Fanuc TP program (LS listing): 190220_hosenrohr_oV3.ls

/PROG  190220_hosenrohr_oV3
/ATTR
COMMENT	= "19-02-22 10:03:29";
PROG_SIZE	= 0;
DEFAULT_GROUP	= 1, 1, *, *, *;
/APPL
    ARC Welding Equipment: 1, *, *, *, *;
/MN
   1:  CALL HOME_ALL;
   1:  UFRAME_NUM = 1;
   1:  UTOOL_NUM = 3;
   1:  COL GUARD ADJUST 150;
   1:  ! -- Layer/Ebene 97 -- !;
   1:  PR[91] = PR[90];
   1:  PR[GP1:91,1] = PR[GP1:90,1] + 0.151;
   1:  PR[GP1:91,2] = PR[GP1:90,2] + 28.908;
   1:  PR[GP1:91,3] = PR[GP1:90,3] + 59.475;
   1:  !Sicherheitspunkt!;
   1:  PR[92] = PR[91];
   1:  PR[92] = PR[GP1:92,3] + 50;
   1:J PR[92];
   1:  !Schweissanfang anfahren!;
   1:L PR[91] R[100]mm/sec CNT100;
   1:  CALL LASER_DRAHT_START;
   1:  PR[GP1:91,1] = PR[GP1:90,1] + -2.869;
   1:  PR[GP1:91,2] = PR[GP1:90,2] + 29.610;
   1:L PR[91] R[100]mm/sec CNT100;
   1:  PR[GP1:91,1] = PR[GP1:90,1] + -5.863;
   1:  PR[GP1:91,2] = PR[GP1:90,2] + 31.726;
   1:L PR[91] R[100]mm/sec CNT100;
   1:  PR[GP1:91,1] = PR[GP1:90,1] + -7.882;
   1:  PR[GP1:91,2] = PR[GP1:90,2] + 32.782;
   1:L PR[91] R[100]mm/sec CNT100;
   1:  PR[GP1:91,1] = PR[GP1:90,1] + -10.388;
   1:  PR[GP1:91,2] = PR[GP1:90,2] + 33.587;
   1:L PR[91] R[100]mm/sec CNT100;
   1:  PR[GP1:91,1] = PR[GP1:90,1] + -18.640;
   1:  PR[GP1:91,2] = PR[GP1:90,2] + 36.440;
   1:L PR[91] R[100]mm/sec CNT100;
   1:  PR[GP1:91,1] = PR[GP1:90,1] + -21.584;
   1:  PR[GP1:91,2] = PR[GP1:90,2] + 36.825;
   1:L PR[91] R[100]mm/sec CNT100;
   1:  PR[GP1:91,1] = PR[GP1:90,1] + -25.063;
   1:  PR[GP1:91,2] = PR[GP1:90,2] + 36.705;
   1:L PR[91] R[100]mm/sec CNT100;
   1:  PR[GP1:91,1] = PR[GP1:90,1] + -32.430;
   1:  PR[GP1:91,2] = PR[GP1:90,2] + 36.668;
   1:L PR[91] R[100]mm/sec CNT100;
   1:  PR[GP1:91,1] = PR[GP1:90,1] + -36.082;
   1:  PR[GP1:91,2] = PR[GP1:90,2] + 35.880;
   1:L PR[91] R[100]mm/sec CNT100;
   1:  PR[GP1:91,1] = PR[GP1:90,1] + -40.103;
   1:  PR[GP1:91,2] = PR[GP1:90,2] + 34.289;
   1:L PR[91] R[100]mm/sec CNT100;
   1:  PR[GP1:91,1] = PR[GP1:90,1] + -45.491;
   1:  PR[GP1:91,2] = PR[GP1:90,2] + 32.375;
   1:L PR[91] R[100]mm/sec CNT100;
   1:  PR[GP1:91,1] = PR[GP1:90,1] + -49.284;
   1:  PR[GP1:91,2] = PR[GP1:90,2] + 30.013;
   1:L PR[91] R[100]mm/sec CNT100;
   1:  PR[GP1:91,1] = PR[GP1:90,1] + -52.981;
   1:  PR[GP1:91,2] = PR[GP1:90,2] + 26.730;
   1:L PR[91] R[100]mm/sec CNT100;
   1:  PR[GP1:91,1] = PR[GP1:90,1] + -56.222;
   1:  PR[GP1:91,2] = PR[GP1:90,2] + 24.107;
   1:L PR[91] R[100]mm/sec CNT100;
   1:  PR[GP1:91,1] = PR[GP1:90,1] + -59.230;
   1:  PR[GP1:91,2] = PR[GP1:90,2] + 20.191;
   1:L PR[91] R[100]mm/sec CNT100;
   1:  PR[GP1:91,1] = PR[GP1:90,1] + -61.763;
   1:  PR[GP1:91,2] = PR[GP1:90,2] + 15.278;
   1:L PR[91] R[100]mm/sec CNT100;
   1:  PR[GP1:91,1] = PR[GP1:90,1] + -63.337;
   1:  PR[GP1:91,2] = PR[GP1:90,2] + 12.647;
   1:L PR[91] R[100]mm/sec CNT100;
   1:  PR[GP1:91,1] = PR[GP1:90,1] + -64.791;
   1:  PR[GP1:91,2] = PR[GP1:90,2] + 7.718;
   1:L PR[91] R[100]mm/sec CNT100;
   1:  PR[GP1:91,1] = PR[GP1:90,1] + -65.271;
   1:  PR[GP1:91,2] = PR[GP1:90,2] + 2.470;
   1:L PR[91] R[100]mm/sec CNT100;
   1:  PR[GP1:91,1] = PR[GP1:90,1] + -65.744;
   1:  PR[GP1:91,2] = PR[GP1:90,2] + -0.100;
   1:L PR[91] R[100]mm/sec CNT100;
   1:  PR[GP1:91,1] = PR[GP1:90,1] + -65.280;
   1:  PR[GP1:91,2] = PR[GP1:90,2] + -5.239;
   1:L PR[91] R[100]mm/sec CNT100;
   1:  PR[GP1:91,1] = PR[GP1:90,1] + -64.798;
   1:  PR[GP1:91,2] = PR[GP1:90,2] + -7.836;
   1:L PR[91] R[100]mm/sec CNT100;
   1:  PR[GP1:91,1] = PR[GP1:90,1] + -63.331;
   1:  PR[GP1:91,2] = PR[GP1:90,2] + -12.812;
   1:L PR[91] R[100]mm/sec CNT100;
   1:  PR[GP1:91,1] = PR[GP1:90,1] + -60.959;
   1:  PR[GP1:91,2] = PR[GP1:90,2] + -17.463;
   1:L PR[91] R[100]mm/sec CNT100;
   1:  PR[GP1:91,1] = PR[GP1:90,1] + -59.241;
   1:  PR[GP1:91,2] = PR[GP1:90,2] + -20.321;
   1:L PR[91] R[100]mm/sec CNT100;
   1:  PR[GP1:91,1] = PR[GP1:90,1] + -56.211;
   1:  PR[GP1:91,2] = PR[GP1:90,2] + -24.265;
   1:L PR[91] R[100]mm/sec CNT100;
   1:  PR[GP1:91,1] = PR[GP1:90,1] + -52.808;
   1:  PR[GP1:91,2] = PR[GP1:90,2] + -27.318;
   1:L PR[91] R[100]mm/sec CNT100;
   1:  PR[GP1:91,1] = PR[GP1:90,1] + -49.292;
   1:  PR[GP1:91,2] = PR[GP1:90,2] + -30.151;
   1:L PR[91] R[100]mm/sec CNT100;
   1:  PR[GP1:91,1] = PR[GP1:90,1] + -45.477;
   1:  PR[GP1:91,2] = PR[GP1:90,2] + -32.528;
   1:L PR[91] R[100]mm/sec CNT100;
   1:  PR[GP1:91,1] = PR[GP1:90,1] + -41.746;
   1:  PR[GP1:91,2] = PR[GP1:90,2] + -34.026;
   1:L PR[91] R[100]mm/sec CNT100;
   1:  PR[GP1:91,1] = PR[GP1:90,1] + -36.085;
   1:  PR[GP1:91,2] = PR[GP1:90,2] + -36.024;
   1:L PR[91] R[100]mm/sec CNT100;
   1:  PR[GP1:91,1] = PR[GP1:90,1] + -32.412;
   1:  PR[GP1:91,2] = PR[GP1:90,2] + -36.816;
   1:L PR[91] R[100]mm/sec CNT100;
   1:  PR[GP1:91,1] = PR[GP1:90,1] + -29.081;
   1:  PR[GP1:91,2] = PR[GP1:90,2] + -36.944;
   1:L PR[91] R[100]mm/sec CNT100;
   1:  PR[GP1:91,1] = PR[GP1:90,1] + -21.580;
   1:  PR[GP1:91,2] = PR[GP1:90,2] + -36.968;
   1:L PR[91] R[100]mm/sec CNT100;
   1:  PR[GP1:91,1] = PR[GP1:90,1] + -18.619;
   1:  PR[GP1:91,2] = PR[GP1:90,2] + -36.581;
   1:L PR[91] R[100]mm/sec CNT100;
   1:  PR[GP1:91,1] = PR[GP1:90,1] + -16.078;
   1:  PR[GP1:91,2] = PR[GP1:90,2] + -35.772;
   1:L PR[91] R[100]mm/sec CNT100;
   1:  PR[GP1:91,1] = PR[GP1:90,1] + -7.875;
   1:  PR[GP1:91,2] = PR[GP1:90,2] + -32.922;
   1:L PR[91] R[100]mm/sec CNT100;
   1:  PR[GP1:91,1] = PR[GP1:90,1] + -5.858;
   1:  PR[GP1:91,2] = PR[GP1:90,2] + -31.867;
   1:L PR[91] R[100]mm/sec CNT100;
   1:  PR[GP1:91,1] = PR[GP1:90,1] + -2.826;
   1:  PR[GP1:91,2] = PR[GP1:90,2] + -29.664;
   1:L PR[91] R[100]mm/sec CNT100;
   1:  PR[GP1:91,1] = PR[GP1:90,1] + -1.739;
   1:  PR[GP1:91,2] = PR[GP1:90,2] + -29.620;
   1:L PR[91] R[100]mm/sec CNT100;
   1:  PR[GP1:91,1] = PR[GP1:90,1] + 1.633;
   1:  PR[GP1:91,2] = PR[GP1:90,2] + -28.901;
   1:L PR[91] R[100]mm/sec CNT100;
   1:  PR[GP1:91,1] = PR[GP1:90,1] + 1.930;
   1:  PR[GP1:91,2] = PR[GP1:90,2] + -29.139;
   1:L PR[91] R[100]mm/sec CNT100;
   1:  PR[GP1:91,1] = PR[GP1:90,1] + 3.140;
   1:  PR[GP1:91,2] = PR[GP1:90,2] + -29.742;
   1:L PR[91] R[100]mm/sec CNT100;
   1:  PR[GP1:91,1] = PR[GP1:90,1] + 6.073;
   1:  PR[GP1:91,2] = PR[GP1:90,2] + -31.873;
   1:L PR[91] R[100]mm/sec CNT100;
   1:  PR[GP1:91,1] = PR[GP1:90,1] + 8.070;
   1:  PR[GP1:91,2] = PR[GP1:90,2] + -32.915;
   1:L PR[91] R[100]mm/sec CNT100;
   1:  PR[GP1:91,1] = PR[GP1:90,1] + 10.573;
   1:  PR[GP1:91,2] = PR[GP1:90,2] + -33.719;
   1:L PR[91] R[100]mm/sec CNT100;
   1:  PR[GP1:91,1] = PR[GP1:90,1] + 18.836;
   1:  PR[GP1:91,2] = PR[GP1:90,2] + -36.580;
   1:L PR[91] R[100]mm/sec CNT100;
   1:  PR[GP1:91,1] = PR[GP1:90,1] + 21.776;
   1:  PR[GP1:91,2] = PR[GP1:90,2] + -36.966;
   1:L PR[91] R[100]mm/sec CNT100;
   1:  PR[GP1:91,1] = PR[GP1:90,1] + 25.238;
   1:  PR[GP1:91,2] = PR[GP1:90,2] + -36.850;
   1:L PR[91] R[100]mm/sec CNT100;
   1:  PR[GP1:91,1] = PR[GP1:90,1] + 32.611;
   1:  PR[GP1:91,2] = PR[GP1:90,2] + -36.818;
   1:L PR[91] R[100]mm/sec CNT100;
   1:  PR[GP1:91,1] = PR[GP1:90,1] + 36.258;
   1:  PR[GP1:91,2] = PR[GP1:90,2] + -36.033;
   1:L PR[91] R[100]mm/sec CNT100;
   1:  PR[GP1:91,1] = PR[GP1:90,1] + 40.284;
   1:  PR[GP1:91,2] = PR[GP1:90,2] + -34.446;
   1:L PR[91] R[100]mm/sec CNT100;
   1:  PR[GP1:91,1] = PR[GP1:90,1] + 45.678;
   1:  PR[GP1:91,2] = PR[GP1:90,2] + -32.535;
   1:L PR[91] R[100]mm/sec CNT100;
   1:  PR[GP1:91,1] = PR[GP1:90,1] + 49.447;
   1:  PR[GP1:91,2] = PR[GP1:90,2] + -30.198;
   1:L PR[91] R[100]mm/sec CNT100;
   1:  PR[GP1:91,1] = PR[GP1:90,1] + 53.124;
   1:  PR[GP1:91,2] = PR[GP1:90,2] + -26.943;
   1:L PR[91] R[100]mm/sec CNT100;
   1:  PR[GP1:91,1] = PR[GP1:90,1] + 56.372;
   1:  PR[GP1:91,2] = PR[GP1:90,2] + -24.313;
   1:L PR[91] R[100]mm/sec CNT100;
   1:  PR[GP1:91,1] = PR[GP1:90,1] + 59.412;
   1:  PR[GP1:91,2] = PR[GP1:90,2] + -20.367;
   1:L PR[91] R[100]mm/sec CNT100;
   1:  PR[GP1:91,1] = PR[GP1:90,1] + 61.952;
   1:  PR[GP1:91,2] = PR[GP1:90,2] + -15.494;
   1:L PR[91] R[100]mm/sec CNT100;
   1:  PR[GP1:91,1] = PR[GP1:90,1] + 63.529;
   1:  PR[GP1:91,2] = PR[GP1:90,2] + -12.866;
   1:L PR[91] R[100]mm/sec CNT100;
   1:  PR[GP1:91,1] = PR[GP1:90,1] + 64.980;
   1:  PR[GP1:91,2] = PR[GP1:90,2] + -8.010;
   1:L PR[91] R[100]mm/sec CNT100;
   1:  PR[GP1:91,1] = PR[GP1:90,1] + 65.484;
   1:  PR[GP1:91,2] = PR[GP1:90,2] + -2.618;
   1:L PR[91] R[100]mm/sec CNT100;
   1:  PR[GP1:91,1] = PR[GP1:90,1] + 65.958;
   1:  PR[GP1:91,2] = PR[GP1:90,2] + -0.045;
   1:L PR[91] R[100]mm/sec CNT100;
   1:  PR[GP1:91,1] = PR[GP1:90,1] + 65.470;
   1:  PR[GP1:91,2] = PR[GP1:90,2] + 5.238;
   1:L PR[91] R[100]mm/sec CNT100;
   1:  PR[GP1:91,1] = PR[GP1:90,1] + 64.988;
   1:  PR[GP1:91,2] = PR[GP1:90,2] + 7.839;
   1:L PR[91] R[100]mm/sec CNT100;
   1:  PR[GP1:91,1] = PR[GP1:90,1] + 63.524;
   1:  PR[GP1:91,2] = PR[GP1:90,2] + 12.740;
   1:L PR[91] R[100]mm/sec CNT100;
   1:  PR[GP1:91,1] = PR[GP1:90,1] + 61.144;
   1:  PR[GP1:91,2] = PR[GP1:90,2] + 17.351;
   1:L PR[91] R[100]mm/sec CNT100;
   1:  PR[GP1:91,1] = PR[GP1:90,1] + 59.425;
   1:  PR[GP1:91,2] = PR[GP1:90,2] + 20.207;
   1:L PR[91] R[100]mm/sec CNT100;
   1:  PR[GP1:91,1] = PR[GP1:90,1] + 56.365;
   1:  PR[GP1:91,2] = PR[GP1:90,2] + 24.179;
   1:L PR[91] R[100]mm/sec CNT100;
   1:  PR[GP1:91,1] = PR[GP1:90,1] + 52.980;
   1:  PR[GP1:91,2] = PR[GP1:90,2] + 27.206;
   1:L PR[91] R[100]mm/sec CNT100;
   1:  PR[GP1:91,1] = PR[GP1:90,1] + 49.463;
   1:  PR[GP1:91,2] = PR[GP1:90,2] + 30.045;
   1:L PR[91] R[100]mm/sec CNT100;
   1:  PR[GP1:91,1] = PR[GP1:90,1] + 45.672;
   1:  PR[GP1:91,2] = PR[GP1:90,2] + 32.395;
   1:L PR[91] R[100]mm/sec CNT100;
   1:  PR[GP1:91,1] = PR[GP1:90,1] + 41.936;
   1:  PR[GP1:91,2] = PR[GP1:90,2] + 33.887;
   1:L PR[91] R[100]mm/sec CNT100;
   1:  PR[GP1:91,1] = PR[GP1:90,1] + 36.277;
   1:  PR[GP1:91,2] = PR[GP1:90,2] + 35.885;
   1:L PR[91] R[100]mm/sec CNT100;
   1:  PR[GP1:91,1] = PR[GP1:90,1] + 32.610;
   1:  PR[GP1:91,2] = PR[GP1:90,2] + 36.674;
   1:L PR[91] R[100]mm/sec CNT100;
   1:  PR[GP1:91,1] = PR[GP1:90,1] + 29.295;
   1:  PR[GP1:91,2] = PR[GP1:90,2] + 36.799;
   1:L PR[91] R[100]mm/sec CNT100;
   1:  PR[GP1:91,1] = PR[GP1:90,1] + 21.797;
   1:  PR[GP1:91,2] = PR[GP1:90,2] + 36.826;
   1:L PR[91] R[100]mm/sec CNT100;
   1:  PR[GP1:91,1] = PR[GP1:90,1] + 18.841;
   1:  PR[GP1:91,2] = PR[GP1:90,2] + 36.437;
   1:L PR[91] R[100]mm/sec CNT100;
   1:  PR[GP1:91,1] = PR[GP1:90,1] + 16.296;
   1:  PR[GP1:91,2] = PR[GP1:90,2] + 35.627;
   1:L PR[91] R[100]mm/sec CNT100;
   1:  PR[GP1:91,1] = PR[GP1:90,1] + 8.090;
   1:  PR[GP1:91,2] = PR[GP1:90,2] + 32.782;
   1:L PR[91] R[100]mm/sec CNT100;
   1:  PR[GP1:91,1] = PR[GP1:90,1] + 6.077;
   1:  PR[GP1:91,2] = PR[GP1:90,2] + 31.732;
   1:L PR[91] R[100]mm/sec CNT100;
   1:  PR[GP1:91,1] = PR[GP1:90,1] + 3.442;
   1:  PR[GP1:91,2] = PR[GP1:90,2] + 29.870;
   1:L PR[91] R[100]mm/sec CNT100;
   1:  PR[GP1:91,1] = PR[GP1:90,1] + 3.445;
   1:  PR[GP1:91,2] = PR[GP1:90,2] + 29.810;
   1:L PR[91] R[100]mm/sec CNT100;
   1:  PR[GP1:91,1] = PR[GP1:90,1] + 1.610;
   1:  PR[GP1:91,2] = PR[GP1:90,2] + 28.789;
   1:L PR[91] R[100]mm/sec CNT100;
   1:  ! -- Layer/Ebene 98 -- !;
   1:  PR[91] = PR[90];
   1:  PR[GP1:91,1] = PR[GP1:90,1] + 0.001;
   1:  PR[GP1:91,2] = PR[GP1:90,2] + 29.166;
   1:  PR[GP1:91,3] = PR[GP1:90,3] + 60.085;
   1:L PR[91] R[100]mm/sec CNT100;
   1:  PR[GP1:91,1] = PR[GP1:90,1] + -2.841;
   1:  PR[GP1:91,2] = PR[GP1:90,2] + 29.827;
   1:L PR[91] R[100]mm/sec CNT100;
   1:  PR[GP1:91,1] = PR[GP1:90,1] + -5.652;
   1:  PR[GP1:91,2] = PR[GP1:90,2] + 31.813;
   1:L PR[91] R[100]mm/sec CNT100;
   1:  PR[GP1:91,1] = PR[GP1:90,1] + -7.540;
   1:  PR[GP1:91,2] = PR[GP1:90,2] + 32.801;
   1:L PR[91] R[100]mm/sec CNT100;
   1:  PR[GP1:91,1] = PR[GP1:90,1] + -9.887;
   1:  PR[GP1:91,2] = PR[GP1:90,2] + 33.555;
   1:L PR[91] R[100]mm/sec CNT100;
   1:  PR[GP1:91,1] = PR[GP1:90,1] + -18.441;
   1:  PR[GP1:91,2] = PR[GP1:90,2] + 36.512;
   1:L PR[91] R[100]mm/sec CNT100;
   1:  PR[GP1:91,1] = PR[GP1:90,1] + -21.232;
   1:  PR[GP1:91,2] = PR[GP1:90,2] + 36.877;
   1:L PR[91] R[100]mm/sec CNT100;
   1:  PR[GP1:91,1] = PR[GP1:90,1] + -24.535;
   1:  PR[GP1:91,2] = PR[GP1:90,2] + 36.764;
   1:L PR[91] R[100]mm/sec CNT100;
   1:  PR[GP1:91,1] = PR[GP1:90,1] + -32.243;
   1:  PR[GP1:91,2] = PR[GP1:90,2] + 36.725;
   1:L PR[91] R[100]mm/sec CNT100;
   1:  PR[GP1:91,1] = PR[GP1:90,1] + -35.737;
   1:  PR[GP1:91,2] = PR[GP1:90,2] + 35.971;
   1:L PR[91] R[100]mm/sec CNT100;
   1:  PR[GP1:91,1] = PR[GP1:90,1] + -39.587;
   1:  PR[GP1:91,2] = PR[GP1:90,2] + 34.447;
   1:L PR[91] R[100]mm/sec CNT100;
   1:  PR[GP1:91,1] = PR[GP1:90,1] + -45.308;
   1:  PR[GP1:91,2] = PR[GP1:90,2] + 32.415;
   1:L PR[91] R[100]mm/sec CNT100;
   1:  PR[GP1:91,1] = PR[GP1:90,1] + -48.959;
   1:  PR[GP1:91,2] = PR[GP1:90,2] + 30.141;
   1:L PR[91] R[100]mm/sec CNT100;
   1:  PR[GP1:91,1] = PR[GP1:90,1] + -52.521;
   1:  PR[GP1:91,2] = PR[GP1:90,2] + 26.978;
   1:L PR[91] R[100]mm/sec CNT100;
   1:  PR[GP1:91,1] = PR[GP1:90,1] + -56.039;
   1:  PR[GP1:91,2] = PR[GP1:90,2] + 24.131;
   1:L PR[91] R[100]mm/sec CNT100;
   1:  PR[GP1:91,1] = PR[GP1:90,1] + -58.946;
   1:  PR[GP1:91,2] = PR[GP1:90,2] + 20.347;
   1:L PR[91] R[100]mm/sec CNT100;
   1:  PR[GP1:91,1] = PR[GP1:90,1] + -61.394;
   1:  PR[GP1:91,2] = PR[GP1:90,2] + 15.596;
   1:L PR[91] R[100]mm/sec CNT100;
   1:  PR[GP1:91,1] = PR[GP1:90,1] + -63.150;
   1:  PR[GP1:91,2] = PR[GP1:90,2] + 12.663;
   1:L PR[91] R[100]mm/sec CNT100;
   1:  PR[GP1:91,1] = PR[GP1:90,1] + -64.558;
   1:  PR[GP1:91,2] = PR[GP1:90,2] + 7.889;
   1:L PR[91] R[100]mm/sec CNT100;
   1:  PR[GP1:91,1] = PR[GP1:90,1] + -65.023;
   1:  PR[GP1:91,2] = PR[GP1:90,2] + 2.804;
   1:L PR[91] R[100]mm/sec CNT100;
   1:  PR[GP1:91,1] = PR[GP1:90,1] + -65.558;
   1:  PR[GP1:91,2] = PR[GP1:90,2] + -0.100;
   1:L PR[91] R[100]mm/sec CNT100;
   1:  PR[GP1:91,1] = PR[GP1:90,1] + -65.108;
   1:  PR[GP1:91,2] = PR[GP1:90,2] + -5.083;
   1:L PR[91] R[100]mm/sec CNT100;
   1:  PR[GP1:91,1] = PR[GP1:90,1] + -64.565;
   1:  PR[GP1:91,2] = PR[GP1:90,2] + -8.007;
   1:L PR[91] R[100]mm/sec CNT100;
   1:  PR[GP1:91,1] = PR[GP1:90,1] + -63.144;
   1:  PR[GP1:91,2] = PR[GP1:90,2] + -12.827;
   1:L PR[91] R[100]mm/sec CNT100;
   1:  PR[GP1:91,1] = PR[GP1:90,1] + -60.846;
   1:  PR[GP1:91,2] = PR[GP1:90,2] + -17.333;
   1:L PR[91] R[100]mm/sec CNT100;
   1:  PR[GP1:91,1] = PR[GP1:90,1] + -58.956;
   1:  PR[GP1:91,2] = PR[GP1:90,2] + -20.478;
   1:L PR[91] R[100]mm/sec CNT100;
   1:  PR[GP1:91,1] = PR[GP1:90,1] + -56.028;
   1:  PR[GP1:91,2] = PR[GP1:90,2] + -24.290;
   1:L PR[91] R[100]mm/sec CNT100;
   1:  PR[GP1:91,1] = PR[GP1:90,1] + -52.738;
   1:  PR[GP1:91,2] = PR[GP1:90,2] + -27.241;
   1:L PR[91] R[100]mm/sec CNT100;
   1:  PR[GP1:91,1] = PR[GP1:90,1] + -48.967;
   1:  PR[GP1:91,2] = PR[GP1:90,2] + -30.280;
   1:L PR[91] R[100]mm/sec CNT100;
   1:  PR[GP1:91,1] = PR[GP1:90,1] + -45.293;
   1:  PR[GP1:91,2] = PR[GP1:90,2] + -32.568;
   1:L PR[91] R[100]mm/sec CNT100;
   1:  PR[GP1:91,1] = PR[GP1:90,1] + -41.700;
   1:  PR[GP1:91,2] = PR[GP1:90,2] + -34.011;
   1:L PR[91] R[100]mm/sec CNT100;
   1:  PR[GP1:91,1] = PR[GP1:90,1] + -35.739;
   1:  PR[GP1:91,2] = PR[GP1:90,2] + -36.114;
   1:L PR[91] R[100]mm/sec CNT100;
   1:  PR[GP1:91,1] = PR[GP1:90,1] + -32.224;
   1:  PR[GP1:91,2] = PR[GP1:90,2] + -36.873;
   1:L PR[91] R[100]mm/sec CNT100;
   1:  PR[GP1:91,1] = PR[GP1:90,1] + -29.035;
   1:  PR[GP1:91,2] = PR[GP1:90,2] + -36.995;
   1:L PR[91] R[100]mm/sec CNT100;
   1:  PR[GP1:91,1] = PR[GP1:90,1] + -21.228;
   1:  PR[GP1:91,2] = PR[GP1:90,2] + -37.020;
   1:L PR[91] R[100]mm/sec CNT100;
   1:  PR[GP1:91,1] = PR[GP1:90,1] + -18.420;
   1:  PR[GP1:91,2] = PR[GP1:90,2] + -36.653;
   1:L PR[91] R[100]mm/sec CNT100;
   1:  PR[GP1:91,1] = PR[GP1:90,1] + -16.010;
   1:  PR[GP1:91,2] = PR[GP1:90,2] + -35.886;
   1:L PR[91] R[100]mm/sec CNT100;
   1:  PR[GP1:91,1] = PR[GP1:90,1] + -7.532;
   1:  PR[GP1:91,2] = PR[GP1:90,2] + -32.940;
   1:L PR[91] R[100]mm/sec CNT100;
   1:  PR[GP1:91,1] = PR[GP1:90,1] + -5.647;
   1:  PR[GP1:91,2] = PR[GP1:90,2] + -31.954;
   1:L PR[91] R[100]mm/sec CNT100;
   1:  PR[GP1:91,1] = PR[GP1:90,1] + -2.798;
   1:  PR[GP1:91,2] = PR[GP1:90,2] + -29.884;
   1:L PR[91] R[100]mm/sec CNT100;
   1:  PR[GP1:91,1] = PR[GP1:90,1] + -1.573;
   1:  PR[GP1:91,2] = PR[GP1:90,2] + -29.835;
   1:L PR[91] R[100]mm/sec CNT100;
   1:  PR[GP1:91,1] = PR[GP1:90,1] + 1.664;
   1:  PR[GP1:91,2] = PR[GP1:90,2] + -29.144;
   1:L PR[91] R[100]mm/sec CNT100;
   1:  PR[GP1:91,1] = PR[GP1:90,1] + 1.978;
   1:  PR[GP1:91,2] = PR[GP1:90,2] + -29.398;
   1:L PR[91] R[100]mm/sec CNT100;
   1:  PR[GP1:91,1] = PR[GP1:90,1] + 3.112;
   1:  PR[GP1:91,2] = PR[GP1:90,2] + -29.962;
   1:L PR[91] R[100]mm/sec CNT100;
   1:  PR[GP1:91,1] = PR[GP1:90,1] + 5.861;
   1:  PR[GP1:91,2] = PR[GP1:90,2] + -31.959;
   1:L PR[91] R[100]mm/sec CNT100;
   1:  PR[GP1:91,1] = PR[GP1:90,1] + 7.728;
   1:  PR[GP1:91,2] = PR[GP1:90,2] + -32.934;
   1:L PR[91] R[100]mm/sec CNT100;
   1:  PR[GP1:91,1] = PR[GP1:90,1] + 10.072;
   1:  PR[GP1:91,2] = PR[GP1:90,2] + -33.686;
   1:L PR[91] R[100]mm/sec CNT100;
   1:  PR[GP1:91,1] = PR[GP1:90,1] + 18.637;
   1:  PR[GP1:91,2] = PR[GP1:90,2] + -36.652;
   1:L PR[91] R[100]mm/sec CNT100;
   1:  PR[GP1:91,1] = PR[GP1:90,1] + 21.424;
   1:  PR[GP1:91,2] = PR[GP1:90,2] + -37.018;
   1:L PR[91] R[100]mm/sec CNT100;
   1:  PR[GP1:91,1] = PR[GP1:90,1] + 24.711;
   1:  PR[GP1:91,2] = PR[GP1:90,2] + -36.908;
   1:L PR[91] R[100]mm/sec CNT100;
   1:  PR[GP1:91,1] = PR[GP1:90,1] + 32.424;
   1:  PR[GP1:91,2] = PR[GP1:90,2] + -36.874;
   1:L PR[91] R[100]mm/sec CNT100;
   1:  PR[GP1:91,1] = PR[GP1:90,1] + 35.913;
   1:  PR[GP1:91,2] = PR[GP1:90,2] + -36.123;
   1:L PR[91] R[100]mm/sec CNT100;
   1:  PR[GP1:91,1] = PR[GP1:90,1] + 39.769;
   1:  PR[GP1:91,2] = PR[GP1:90,2] + -34.604;
   1:L PR[91] R[100]mm/sec CNT100;
   1:  PR[GP1:91,1] = PR[GP1:90,1] + 45.495;
   1:  PR[GP1:91,2] = PR[GP1:90,2] + -32.575;
   1:L PR[91] R[100]mm/sec CNT100;
   1:  PR[GP1:91,1] = PR[GP1:90,1] + 49.124;
   1:  PR[GP1:91,2] = PR[GP1:90,2] + -30.325;
   1:L PR[91] R[100]mm/sec CNT100;
   1:  PR[GP1:91,1] = PR[GP1:90,1] + 52.666;
   1:  PR[GP1:91,2] = PR[GP1:90,2] + -27.189;
   1:L PR[91] R[100]mm/sec CNT100;
   1:  PR[GP1:91,1] = PR[GP1:90,1] + 56.191;
   1:  PR[GP1:91,2] = PR[GP1:90,2] + -24.336;
   1:L PR[91] R[100]mm/sec CNT100;
   1:  PR[GP1:91,1] = PR[GP1:90,1] + 59.128;
   1:  PR[GP1:91,2] = PR[GP1:90,2] + -20.522;
   1:L PR[91] R[100]mm/sec CNT100;
   1:  PR[GP1:91,1] = PR[GP1:90,1] + 61.584;
   1:  PR[GP1:91,2] = PR[GP1:90,2] + -15.809;
   1:L PR[91] R[100]mm/sec CNT100;
   1:  PR[GP1:91,1] = PR[GP1:90,1] + 63.343;
   1:  PR[GP1:91,2] = PR[GP1:90,2] + -12.880;
   1:L PR[91] R[100]mm/sec CNT100;
   1:  PR[GP1:91,1] = PR[GP1:90,1] + 64.748;
   1:  PR[GP1:91,2] = PR[GP1:90,2] + -8.177;
   1:L PR[91] R[100]mm/sec CNT100;
   1:  PR[GP1:91,1] = PR[GP1:90,1] + 65.236;
   1:  PR[GP1:91,2] = PR[GP1:90,2] + -2.953;
   1:L PR[91] R[100]mm/sec CNT100;
   1:  PR[GP1:91,1] = PR[GP1:90,1] + 65.771;
   1:  PR[GP1:91,2] = PR[GP1:90,2] + -0.045;
   1:L PR[91] R[100]mm/sec CNT100;
   1:  PR[GP1:91,1] = PR[GP1:90,1] + 65.299;
   1:  PR[GP1:91,2] = PR[GP1:90,2] + 5.077;
   1:L PR[91] R[100]mm/sec CNT100;
   1:  PR[GP1:91,1] = PR[GP1:90,1] + 64.756;
   1:  PR[GP1:91,2] = PR[GP1:90,2] + 8.006;
   1:L PR[91] R[100]mm/sec CNT100;
   1:  PR[GP1:91,1] = PR[GP1:90,1] + 63.337;
   1:  PR[GP1:91,2] = PR[GP1:90,2] + 12.754;
   1:L PR[91] R[100]mm/sec CNT100;
   1:  PR[GP1:91,1] = PR[GP1:90,1] + 61.032;
   1:  PR[GP1:91,2] = PR[GP1:90,2] + 17.221;
   1:L PR[91] R[100]mm/sec CNT100;
   1:  PR[GP1:91,1] = PR[GP1:90,1] + 59.141;
   1:  PR[GP1:91,2] = PR[GP1:90,2] + 20.361;
   1:L PR[91] R[100]mm/sec CNT100;
   1:  PR[GP1:91,1] = PR[GP1:90,1] + 56.183;
   1:  PR[GP1:91,2] = PR[GP1:90,2] + 24.201;
   1:L PR[91] R[100]mm/sec CNT100;
   1:  PR[GP1:91,1] = PR[GP1:90,1] + 52.911;
   1:  PR[GP1:91,2] = PR[GP1:90,2] + 27.127;
   1:L PR[91] R[100]mm/sec CNT100;
   1:  PR[GP1:91,1] = PR[GP1:90,1] + 49.140;
   1:  PR[GP1:91,2] = PR[GP1:90,2] + 30.172;
   1:L PR[91] R[100]mm/sec CNT100;
   1:  PR[GP1:91,1] = PR[GP1:90,1] + 45.490;
   1:  PR[GP1:91,2] = PR[GP1:90,2] + 32.434;
   1:L PR[91] R[100]mm/sec CNT100;
   1:  PR[GP1:91,1] = PR[GP1:90,1] + 41.892;
   1:  PR[GP1:91,2] = PR[GP1:90,2] + 33.871;
   1:L PR[91] R[100]mm/sec CNT100;
   1:  PR[GP1:91,1] = PR[GP1:90,1] + 35.932;
   1:  PR[GP1:91,2] = PR[GP1:90,2] + 35.975;
   1:L PR[91] R[100]mm/sec CNT100;
   1:  PR[GP1:91,1] = PR[GP1:90,1] + 32.423;
   1:  PR[GP1:91,2] = PR[GP1:90,2] + 36.731;
   1:L PR[91] R[100]mm/sec CNT100;
   1:  PR[GP1:91,1] = PR[GP1:90,1] + 29.250;
   1:  PR[GP1:91,2] = PR[GP1:90,2] + 36.850;
   1:L PR[91] R[100]mm/sec CNT100;
   1:  PR[GP1:91,1] = PR[GP1:90,1] + 21.446;
   1:  PR[GP1:91,2] = PR[GP1:90,2] + 36.878;
   1:L PR[91] R[100]mm/sec CNT100;
   1:  PR[GP1:91,1] = PR[GP1:90,1] + 18.642;
   1:  PR[GP1:91,2] = PR[GP1:90,2] + 36.509;
   1:L PR[91] R[100]mm/sec CNT100;
   1:  PR[GP1:91,1] = PR[GP1:90,1] + 16.228;
   1:  PR[GP1:91,2] = PR[GP1:90,2] + 35.741;
   1:L PR[91] R[100]mm/sec CNT100;
   1:  PR[GP1:91,1] = PR[GP1:90,1] + 7.748;
   1:  PR[GP1:91,2] = PR[GP1:90,2] + 32.801;
   1:L PR[91] R[100]mm/sec CNT100;
   1:  PR[GP1:91,1] = PR[GP1:90,1] + 5.866;
   1:  PR[GP1:91,2] = PR[GP1:90,2] + 31.819;
   1:L PR[91] R[100]mm/sec CNT100;
   1:  PR[GP1:91,1] = PR[GP1:90,1] + 3.414;
   1:  PR[GP1:91,2] = PR[GP1:90,2] + 30.086;
   1:L PR[91] R[100]mm/sec CNT100;
   1:  PR[GP1:91,1] = PR[GP1:90,1] + 3.417;
   1:  PR[GP1:91,2] = PR[GP1:90,2] + 30.021;
   1:L PR[91] R[100]mm/sec CNT100;
   1:  PR[GP1:91,1] = PR[GP1:90,1] + 1.640;
   1:  PR[GP1:91,2] = PR[GP1:90,2] + 29.032;
   1:L PR[91] R[100]mm/sec CNT100;
   1:  ! -- Layer/Ebene 99 -- !;
   1:  PR[91] = PR[90];
   1:  PR[GP1:91,1] = PR[GP1:90,1] + -0.150;
   1:  PR[GP1:91,2] = PR[GP1:90,2] + 29.425;
   1:  PR[GP1:91,3] = PR[GP1:90,3] + 60.695;
   1:L PR[91] R[100]mm/sec CNT100;
   1:  PR[GP1:91,1] = PR[GP1:90,1] + -2.813;
   1:  PR[GP1:91,2] = PR[GP1:90,2] + 30.043;
   1:L PR[91] R[100]mm/sec CNT100;
   1:  PR[GP1:91,1] = PR[GP1:90,1] + -5.441;
   1:  PR[GP1:91,2] = PR[GP1:90,2] + 31.901;
   1:L PR[91] R[100]mm/sec CNT100;
   1:  PR[GP1:91,1] = PR[GP1:90,1] + -7.199;
   1:  PR[GP1:91,2] = PR[GP1:90,2] + 32.820;
   1:L PR[91] R[100]mm/sec CNT100;
   1:  PR[GP1:91,1] = PR[GP1:90,1] + -9.386;
   1:  PR[GP1:91,2] = PR[GP1:90,2] + 33.523;
   1:L PR[91] R[100]mm/sec CNT100;
   1:  PR[GP1:91,1] = PR[GP1:90,1] + -18.243;
   1:  PR[GP1:91,2] = PR[GP1:90,2] + 36.585;
   1:L PR[91] R[100]mm/sec CNT100;
   1:  PR[GP1:91,1] = PR[GP1:90,1] + -20.881;
   1:  PR[GP1:91,2] = PR[GP1:90,2] + 36.929;
   1:L PR[91] R[100]mm/sec CNT100;
   1:  PR[GP1:91,1] = PR[GP1:90,1] + -24.007;
   1:  PR[GP1:91,2] = PR[GP1:90,2] + 36.822;
   1:L PR[91] R[100]mm/sec CNT100;
   1:  PR[GP1:91,1] = PR[GP1:90,1] + -32.055;
   1:  PR[GP1:91,2] = PR[GP1:90,2] + 36.782;
   1:L PR[91] R[100]mm/sec CNT100;
   1:  PR[GP1:91,1] = PR[GP1:90,1] + -35.391;
   1:  PR[GP1:91,2] = PR[GP1:90,2] + 36.062;
   1:L PR[91] R[100]mm/sec CNT100;
   1:  PR[GP1:91,1] = PR[GP1:90,1] + -39.072;
   1:  PR[GP1:91,2] = PR[GP1:90,2] + 34.605;
   1:L PR[91] R[100]mm/sec CNT100;
   1:  PR[GP1:91,1] = PR[GP1:90,1] + -45.124;
   1:  PR[GP1:91,2] = PR[GP1:90,2] + 32.455;
   1:L PR[91] R[100]mm/sec CNT100;
   1:  PR[GP1:91,1] = PR[GP1:90,1] + -48.634;
   1:  PR[GP1:91,2] = PR[GP1:90,2] + 30.269;
   1:L PR[91] R[100]mm/sec CNT100;
   1:  PR[GP1:91,1] = PR[GP1:90,1] + -52.061;
   1:  PR[GP1:91,2] = PR[GP1:90,2] + 27.227;
   1:L PR[91] R[100]mm/sec CNT100;
   1:  PR[GP1:91,1] = PR[GP1:90,1] + -55.855;
   1:  PR[GP1:91,2] = PR[GP1:90,2] + 24.156;
   1:L PR[91] R[100]mm/sec CNT100;
   1:  PR[GP1:91,1] = PR[GP1:90,1] + -58.661;
   1:  PR[GP1:91,2] = PR[GP1:90,2] + 20.503;
   1:L PR[91] R[100]mm/sec CNT100;
   1:  PR[GP1:91,1] = PR[GP1:90,1] + -61.026;
   1:  PR[GP1:91,2] = PR[GP1:90,2] + 15.914;
   1:L PR[91] R[100]mm/sec CNT100;
   1:  PR[GP1:91,1] = PR[GP1:90,1] + -62.963;
   1:  PR[GP1:91,2] = PR[GP1:90,2] + 12.678;
   1:L PR[91] R[100]mm/sec CNT100;
   1:  PR[GP1:91,1] = PR[GP1:90,1] + -64.324;
   1:  PR[GP1:91,2] = PR[GP1:90,2] + 8.061;
   1:L PR[91] R[100]mm/sec CNT100;
   1:  PR[GP1:91,1] = PR[GP1:90,1] + -64.775;
   1:  PR[GP1:91,2] = PR[GP1:90,2] + 3.139;
   1:L PR[91] R[100]mm/sec CNT100;
   1:  PR[GP1:91,1] = PR[GP1:90,1] + -65.372;
   1:  PR[GP1:91,2] = PR[GP1:90,2] + -0.100;
   1:L PR[91] R[100]mm/sec CNT100;
   1:  PR[GP1:91,1] = PR[GP1:90,1] + -64.936;
   1:  PR[GP1:91,2] = PR[GP1:90,2] + -4.926;
   1:L PR[91] R[100]mm/sec CNT100;
   1:  PR[GP1:91,1] = PR[GP1:90,1] + -64.332;
   1:  PR[GP1:91,2] = PR[GP1:90,2] + -8.179;
   1:L PR[91] R[100]mm/sec CNT100;
   1:  PR[GP1:91,1] = PR[GP1:90,1] + -62.957;
   1:  PR[GP1:91,2] = PR[GP1:90,2] + -12.843;
   1:L PR[91] R[100]mm/sec CNT100;
   1:  PR[GP1:91,1] = PR[GP1:90,1] + -60.733;
   1:  PR[GP1:91,2] = PR[GP1:90,2] + -17.203;
   1:L PR[91] R[100]mm/sec CNT100;
   1:  PR[GP1:91,1] = PR[GP1:90,1] + -58.671;
   1:  PR[GP1:91,2] = PR[GP1:90,2] + -20.634;
   1:L PR[91] R[100]mm/sec CNT100;
   1:  PR[GP1:91,1] = PR[GP1:90,1] + -55.844;
   1:  PR[GP1:91,2] = PR[GP1:90,2] + -24.314;
   1:L PR[91] R[100]mm/sec CNT100;
   1:  PR[GP1:91,1] = PR[GP1:90,1] + -52.667;
   1:  PR[GP1:91,2] = PR[GP1:90,2] + -27.163;
   1:L PR[91] R[100]mm/sec CNT100;
   1:  PR[GP1:91,1] = PR[GP1:90,1] + -48.642;
   1:  PR[GP1:91,2] = PR[GP1:90,2] + -30.408;
   1:L PR[91] R[100]mm/sec CNT100;
   1:  PR[GP1:91,1] = PR[GP1:90,1] + -45.109;
   1:  PR[GP1:91,2] = PR[GP1:90,2] + -32.609;
   1:L PR[91] R[100]mm/sec CNT100;
   1:  PR[GP1:91,1] = PR[GP1:90,1] + -41.654;
   1:  PR[GP1:91,2] = PR[GP1:90,2] + -33.996;
   1:L PR[91] R[100]mm/sec CNT100;
   1:  PR[GP1:91,1] = PR[GP1:90,1] + -35.393;
   1:  PR[GP1:91,2] = PR[GP1:90,2] + -36.205;
   1:L PR[91] R[100]mm/sec CNT100;
   1:  PR[GP1:91,1] = PR[GP1:90,1] + -32.036;
   1:  PR[GP1:91,2] = PR[GP1:90,2] + -36.929;
   1:L PR[91] R[100]mm/sec CNT100;
   1:  PR[GP1:91,1] = PR[GP1:90,1] + -28.989;
   1:  PR[GP1:91,2] = PR[GP1:90,2] + -37.047;
   1:L PR[91] R[100]mm/sec CNT100;
   1:  PR[GP1:91,1] = PR[GP1:90,1] + -20.876;
   1:  PR[GP1:91,2] = PR[GP1:90,2] + -37.072;
   1:L PR[91] R[100]mm/sec CNT100;
   1:  PR[GP1:91,1] = PR[GP1:90,1] + -18.221;
   1:  PR[GP1:91,2] = PR[GP1:90,2] + -36.725;
   1:L PR[91] R[100]mm/sec CNT100;
   1:  PR[GP1:91,1] = PR[GP1:90,1] + -15.941;
   1:  PR[GP1:91,2] = PR[GP1:90,2] + -36.000;
   1:L PR[91] R[100]mm/sec CNT100;
   1:  PR[GP1:91,1] = PR[GP1:90,1] + -7.190;
   1:  PR[GP1:91,2] = PR[GP1:90,2] + -32.959;
   1:L PR[91] R[100]mm/sec CNT100;
   1:  PR[GP1:91,1] = PR[GP1:90,1] + -5.436;
   1:  PR[GP1:91,2] = PR[GP1:90,2] + -32.041;
   1:L PR[91] R[100]mm/sec CNT100;
   1:  PR[GP1:91,1] = PR[GP1:90,1] + -2.770;
   1:  PR[GP1:91,2] = PR[GP1:90,2] + -30.104;
   1:L PR[91] R[100]mm/sec CNT100;
   1:  PR[GP1:91,1] = PR[GP1:90,1] + -1.407;
   1:  PR[GP1:91,2] = PR[GP1:90,2] + -30.050;
   1:L PR[91] R[100]mm/sec CNT100;
   1:  PR[GP1:91,1] = PR[GP1:90,1] + 1.694;
   1:  PR[GP1:91,2] = PR[GP1:90,2] + -29.388;
   1:L PR[91] R[100]mm/sec CNT100;
   1:  PR[GP1:91,1] = PR[GP1:90,1] + 2.027;
   1:  PR[GP1:91,2] = PR[GP1:90,2] + -29.656;
   1:L PR[91] R[100]mm/sec CNT100;
   1:  PR[GP1:91,1] = PR[GP1:90,1] + 3.084;
   1:  PR[GP1:91,2] = PR[GP1:90,2] + -30.182;
   1:L PR[91] R[100]mm/sec CNT100;
   1:  PR[GP1:91,1] = PR[GP1:90,1] + 5.650;
   1:  PR[GP1:91,2] = PR[GP1:90,2] + -32.046;
   1:L PR[91] R[100]mm/sec CNT100;
   1:  PR[GP1:91,1] = PR[GP1:90,1] + 7.386;
   1:  PR[GP1:91,2] = PR[GP1:90,2] + -32.952;
   1:L PR[91] R[100]mm/sec CNT100;
   1:  PR[GP1:91,1] = PR[GP1:90,1] + 9.570;
   1:  PR[GP1:91,2] = PR[GP1:90,2] + -33.654;
   1:L PR[91] R[100]mm/sec CNT100;
   1:  PR[GP1:91,1] = PR[GP1:90,1] + 18.438;
   1:  PR[GP1:91,2] = PR[GP1:90,2] + -36.724;
   1:L PR[91] R[100]mm/sec CNT100;
   1:  PR[GP1:91,1] = PR[GP1:90,1] + 21.072;
   1:  PR[GP1:91,2] = PR[GP1:90,2] + -37.071;
   1:L PR[91] R[100]mm/sec CNT100;
   1:  PR[GP1:91,1] = PR[GP1:90,1] + 24.183;
   1:  PR[GP1:91,2] = PR[GP1:90,2] + -36.966;
   1:L PR[91] R[100]mm/sec CNT100;
   1:  PR[GP1:91,1] = PR[GP1:90,1] + 32.237;
   1:  PR[GP1:91,2] = PR[GP1:90,2] + -36.931;
   1:L PR[91] R[100]mm/sec CNT100;
   1:  PR[GP1:91,1] = PR[GP1:90,1] + 35.568;
   1:  PR[GP1:91,2] = PR[GP1:90,2] + -36.214;
   1:L PR[91] R[100]mm/sec CNT100;
   1:  PR[GP1:91,1] = PR[GP1:90,1] + 39.253;
   1:  PR[GP1:91,2] = PR[GP1:90,2] + -34.762;
   1:L PR[91] R[100]mm/sec CNT100;
   1:  PR[GP1:91,1] = PR[GP1:90,1] + 45.312;
   1:  PR[GP1:91,2] = PR[GP1:90,2] + -32.614;
   1:L PR[91] R[100]mm/sec CNT100;
   1:  PR[GP1:91,1] = PR[GP1:90,1] + 48.800;
   1:  PR[GP1:91,2] = PR[GP1:90,2] + -30.452;
   1:L PR[91] R[100]mm/sec CNT100;
   1:  PR[GP1:91,1] = PR[GP1:90,1] + 52.207;
   1:  PR[GP1:91,2] = PR[GP1:90,2] + -27.435;
   1:L PR[91] R[100]mm/sec CNT100;
   1:  PR[GP1:91,1] = PR[GP1:90,1] + 56.009;
   1:  PR[GP1:91,2] = PR[GP1:90,2] + -24.358;
   1:L PR[91] R[100]mm/sec CNT100;
   1:  PR[GP1:91,1] = PR[GP1:90,1] + 58.845;
   1:  PR[GP1:91,2] = PR[GP1:90,2] + -20.677;
   1:L PR[91] R[100]mm/sec CNT100;
   1:  PR[GP1:91,1] = PR[GP1:90,1] + 61.217;
   1:  PR[GP1:91,2] = PR[GP1:90,2] + -16.125;
   1:L PR[91] R[100]mm/sec CNT100;
   1:  PR[GP1:91,1] = PR[GP1:90,1] + 63.156;
   1:  PR[GP1:91,2] = PR[GP1:90,2] + -12.894;
   1:L PR[91] R[100]mm/sec CNT100;
   1:  PR[GP1:91,1] = PR[GP1:90,1] + 64.515;
   1:  PR[GP1:91,2] = PR[GP1:90,2] + -8.345;
   1:L PR[91] R[100]mm/sec CNT100;
   1:  PR[GP1:91,1] = PR[GP1:90,1] + 64.988;
   1:  PR[GP1:91,2] = PR[GP1:90,2] + -3.288;
   1:L PR[91] R[100]mm/sec CNT100;
   1:  PR[GP1:91,1] = PR[GP1:90,1] + 65.585;
   1:  PR[GP1:91,2] = PR[GP1:90,2] + -0.045;
   1:L PR[91] R[100]mm/sec CNT100;
   1:  PR[GP1:91,1] = PR[GP1:90,1] + 65.127;
   1:  PR[GP1:91,2] = PR[GP1:90,2] + 4.916;
   1:L PR[91] R[100]mm/sec CNT100;
   1:  PR[GP1:91,1] = PR[GP1:90,1] + 64.523;
   1:  PR[GP1:91,2] = PR[GP1:90,2] + 8.174;
   1:L PR[91] R[100]mm/sec CNT100;
   1:  PR[GP1:91,1] = PR[GP1:90,1] + 63.151;
   1:  PR[GP1:91,2] = PR[GP1:90,2] + 12.768;
   1:L PR[91] R[100]mm/sec CNT100;
   1:  PR[GP1:91,1] = PR[GP1:90,1] + 60.920;
   1:  PR[GP1:91,2] = PR[GP1:90,2] + 17.090;
   1:L PR[91] R[100]mm/sec CNT100;
   1:  PR[GP1:91,1] = PR[GP1:90,1] + 58.858;
   1:  PR[GP1:91,2] = PR[GP1:90,2] + 20.516;
   1:L PR[91] R[100]mm/sec CNT100;
   1:  PR[GP1:91,1] = PR[GP1:90,1] + 56.002;
   1:  PR[GP1:91,2] = PR[GP1:90,2] + 24.224;
   1:L PR[91] R[100]mm/sec CNT100;
   1:  PR[GP1:91,1] = PR[GP1:90,1] + 52.842;
   1:  PR[GP1:91,2] = PR[GP1:90,2] + 27.049;
   1:L PR[91] R[100]mm/sec CNT100;
   1:  PR[GP1:91,1] = PR[GP1:90,1] + 48.817;
   1:  PR[GP1:91,2] = PR[GP1:90,2] + 30.298;
   1:L PR[91] R[100]mm/sec CNT100;
   1:  PR[GP1:91,1] = PR[GP1:90,1] + 45.307;
   1:  PR[GP1:91,2] = PR[GP1:90,2] + 32.474;
   1:L PR[91] R[100]mm/sec CNT100;
   1:  PR[GP1:91,1] = PR[GP1:90,1] + 41.847;
   1:  PR[GP1:91,2] = PR[GP1:90,2] + 33.856;
   1:L PR[91] R[100]mm/sec CNT100;
   1:  PR[GP1:91,1] = PR[GP1:90,1] + 35.588;
   1:  PR[GP1:91,2] = PR[GP1:90,2] + 36.066;
   1:L PR[91] R[100]mm/sec CNT100;
   1:  PR[GP1:91,1] = PR[GP1:90,1] + 32.236;
   1:  PR[GP1:91,2] = PR[GP1:90,2] + 36.787;
   1:L PR[91] R[100]mm/sec CNT100;
   1:  PR[GP1:91,1] = PR[GP1:90,1] + 29.205;
   1:  PR[GP1:91,2] = PR[GP1:90,2] + 36.901;
   1:L PR[91] R[100]mm/sec CNT100;
   1:  PR[GP1:91,1] = PR[GP1:90,1] + 21.095;
   1:  PR[GP1:91,2] = PR[GP1:90,2] + 36.930;
   1:L PR[91] R[100]mm/sec CNT100;
   1:  PR[GP1:91,1] = PR[GP1:90,1] + 18.444;
   1:  PR[GP1:91,2] = PR[GP1:90,2] + 36.581;
   1:L PR[91] R[100]mm/sec CNT100;
   1:  PR[GP1:91,1] = PR[GP1:90,1] + 16.161;
   1:  PR[GP1:91,2] = PR[GP1:90,2] + 35.855;
   1:L PR[91] R[100]mm/sec CNT100;
   1:  PR[GP1:91,1] = PR[GP1:90,1] + 7.407;
   1:  PR[GP1:91,2] = PR[GP1:90,2] + 32.820;
   1:L PR[91] R[100]mm/sec CNT100;
   1:  PR[GP1:91,1] = PR[GP1:90,1] + 5.655;
   1:  PR[GP1:91,2] = PR[GP1:90,2] + 31.906;
   1:L PR[91] R[100]mm/sec CNT100;
   1:  PR[GP1:91,1] = PR[GP1:90,1] + 3.386;
   1:  PR[GP1:91,2] = PR[GP1:90,2] + 30.303;
   1:L PR[91] R[100]mm/sec CNT100;
   1:  PR[GP1:91,1] = PR[GP1:90,1] + 3.390;
   1:  PR[GP1:91,2] = PR[GP1:90,2] + 30.232;
   1:L PR[91] R[100]mm/sec CNT100;
   1:  PR[GP1:91,1] = PR[GP1:90,1] + 1.670;
   1:  PR[GP1:91,2] = PR[GP1:90,2] + 29.275;
   1:L PR[91] R[100]mm/sec CNT100;
   1:  ! -- Layer/Ebene 100 -- !;
   1:  PR[91] = PR[90];
   1:  PR[GP1:91,1] = PR[GP1:90,1] + -0.301;
   1:  PR[GP1:91,2] = PR[GP1:90,2] + 29.683;
   1:  PR[GP1:91,3] = PR[GP1:90,3] + 61.305;
   1:L PR[91] R[100]mm/sec CNT100;
   1:  PR[GP1:91,1] = PR[GP1:90,1] + -2.785;
   1:  PR[GP1:91,2] = PR[GP1:90,2] + 30.260;
   1:L PR[91] R[100]mm/sec CNT100;
   1:  PR[GP1:91,1] = PR[GP1:90,1] + -5.231;
   1:  PR[GP1:91,2] = PR[GP1:90,2] + 31.988;
   1:L PR[91] R[100]mm/sec CNT100;
   1:  PR[GP1:91,1] = PR[GP1:90,1] + -6.857;
   1:  PR[GP1:91,2] = PR[GP1:90,2] + 32.839;
   1:L PR[91] R[100]mm/sec CNT100;
   1:  PR[GP1:91,1] = PR[GP1:90,1] + -8.885;
   1:  PR[GP1:91,2] = PR[GP1:90,2] + 33.490;
   1:L PR[91] R[100]mm/sec CNT100;
   1:  PR[GP1:91,1] = PR[GP1:90,1] + -18.044;
   1:  PR[GP1:91,2] = PR[GP1:90,2] + 36.657;
   1:L PR[91] R[100]mm/sec CNT100;
   1:  PR[GP1:91,1] = PR[GP1:90,1] + -20.529;
   1:  PR[GP1:91,2] = PR[GP1:90,2] + 36.982;
   1:L PR[91] R[100]mm/sec CNT100;
   1:  PR[GP1:91,1] = PR[GP1:90,1] + -23.479;
   1:  PR[GP1:91,2] = PR[GP1:90,2] + 36.880;
   1:L PR[91] R[100]mm/sec CNT100;
   1:  PR[GP1:91,1] = PR[GP1:90,1] + -31.867;
   1:  PR[GP1:91,2] = PR[GP1:90,2] + 36.838;
   1:L PR[91] R[100]mm/sec CNT100;
   1:  PR[GP1:91,1] = PR[GP1:90,1] + -35.046;
   1:  PR[GP1:91,2] = PR[GP1:90,2] + 36.152;
   1:L PR[91] R[100]mm/sec CNT100;
   1:  PR[GP1:91,1] = PR[GP1:90,1] + -38.556;
   1:  PR[GP1:91,2] = PR[GP1:90,2] + 34.763;
   1:L PR[91] R[100]mm/sec CNT100;
   1:  PR[GP1:91,1] = PR[GP1:90,1] + -44.941;
   1:  PR[GP1:91,2] = PR[GP1:90,2] + 32.495;
   1:L PR[91] R[100]mm/sec CNT100;
   1:  PR[GP1:91,1] = PR[GP1:90,1] + -48.309;
   1:  PR[GP1:91,2] = PR[GP1:90,2] + 30.397;
   1:L PR[91] R[100]mm/sec CNT100;
   1:  PR[GP1:91,1] = PR[GP1:90,1] + -51.600;
   1:  PR[GP1:91,2] = PR[GP1:90,2] + 27.475;
   1:L PR[91] R[100]mm/sec CNT100;
   1:  PR[GP1:91,1] = PR[GP1:90,1] + -55.672;
   1:  PR[GP1:91,2] = PR[GP1:90,2] + 24.180;
   1:L PR[91] R[100]mm/sec CNT100;
   1:  PR[GP1:91,1] = PR[GP1:90,1] + -58.377;
   1:  PR[GP1:91,2] = PR[GP1:90,2] + 20.659;
   1:L PR[91] R[100]mm/sec CNT100;
   1:  PR[GP1:91,1] = PR[GP1:90,1] + -60.658;
   1:  PR[GP1:91,2] = PR[GP1:90,2] + 16.232;
   1:L PR[91] R[100]mm/sec CNT100;
   1:  PR[GP1:91,1] = PR[GP1:90,1] + -62.776;
   1:  PR[GP1:91,2] = PR[GP1:90,2] + 12.694;
   1:L PR[91] R[100]mm/sec CNT100;
   1:  PR[GP1:91,1] = PR[GP1:90,1] + -64.091;
   1:  PR[GP1:91,2] = PR[GP1:90,2] + 8.232;
   1:L PR[91] R[100]mm/sec CNT100;
   1:  PR[GP1:91,1] = PR[GP1:90,1] + -64.527;
   1:  PR[GP1:91,2] = PR[GP1:90,2] + 3.473;
   1:L PR[91] R[100]mm/sec CNT100;
   1:  PR[GP1:91,1] = PR[GP1:90,1] + -65.186;
   1:  PR[GP1:91,2] = PR[GP1:90,2] + -0.100;
   1:L PR[91] R[100]mm/sec CNT100;
   1:  PR[GP1:91,1] = PR[GP1:90,1] + -64.764;
   1:  PR[GP1:91,2] = PR[GP1:90,2] + -4.770;
   1:L PR[91] R[100]mm/sec CNT100;
   1:  PR[GP1:91,1] = PR[GP1:90,1] + -64.099;
   1:  PR[GP1:91,2] = PR[GP1:90,2] + -8.351;
   1:L PR[91] R[100]mm/sec CNT100;
   1:  PR[GP1:91,1] = PR[GP1:90,1] + -62.770;
   1:  PR[GP1:91,2] = PR[GP1:90,2] + -12.859;
   1:L PR[91] R[100]mm/sec CNT100;
   1:  PR[GP1:91,1] = PR[GP1:90,1] + -60.620;
   1:  PR[GP1:91,2] = PR[GP1:90,2] + -17.074;
   1:L PR[91] R[100]mm/sec CNT100;
   1:  PR[GP1:91,1] = PR[GP1:90,1] + -58.387;
   1:  PR[GP1:91,2] = PR[GP1:90,2] + -20.790;
   1:L PR[91] R[100]mm/sec CNT100;
   1:  PR[GP1:91,1] = PR[GP1:90,1] + -55.660;
   1:  PR[GP1:91,2] = PR[GP1:90,2] + -24.338;
   1:L PR[91] R[100]mm/sec CNT100;
   1:  PR[GP1:91,1] = PR[GP1:90,1] + -52.597;
   1:  PR[GP1:91,2] = PR[GP1:90,2] + -27.086;
   1:L PR[91] R[100]mm/sec CNT100;
   1:  PR[GP1:91,1] = PR[GP1:90,1] + -48.317;
   1:  PR[GP1:91,2] = PR[GP1:90,2] + -30.536;
   1:L PR[91] R[100]mm/sec CNT100;
   1:  PR[GP1:91,1] = PR[GP1:90,1] + -44.925;
   1:  PR[GP1:91,2] = PR[GP1:90,2] + -32.649;
   1:L PR[91] R[100]mm/sec CNT100;
   1:  PR[GP1:91,1] = PR[GP1:90,1] + -41.608;
   1:  PR[GP1:91,2] = PR[GP1:90,2] + -33.981;
   1:L PR[91] R[100]mm/sec CNT100;
   1:  PR[GP1:91,1] = PR[GP1:90,1] + -35.047;
   1:  PR[GP1:91,2] = PR[GP1:90,2] + -36.296;
   1:L PR[91] R[100]mm/sec CNT100;
   1:  PR[GP1:91,1] = PR[GP1:90,1] + -31.847;
   1:  PR[GP1:91,2] = PR[GP1:90,2] + -36.986;
   1:L PR[91] R[100]mm/sec CNT100;
   1:  PR[GP1:91,1] = PR[GP1:90,1] + -28.944;
   1:  PR[GP1:91,2] = PR[GP1:90,2] + -37.098;
   1:L PR[91] R[100]mm/sec CNT100;
   1:  PR[GP1:91,1] = PR[GP1:90,1] + -20.524;
   1:  PR[GP1:91,2] = PR[GP1:90,2] + -37.124;
   1:L PR[91] R[100]mm/sec CNT100;
   1:  PR[GP1:91,1] = PR[GP1:90,1] + -18.023;
   1:  PR[GP1:91,2] = PR[GP1:90,2] + -36.798;
   1:L PR[91] R[100]mm/sec CNT100;
   1:  PR[GP1:91,1] = PR[GP1:90,1] + -15.873;
   1:  PR[GP1:91,2] = PR[GP1:90,2] + -36.113;
   1:L PR[91] R[100]mm/sec CNT100;
   1:  PR[GP1:91,1] = PR[GP1:90,1] + -6.848;
   1:  PR[GP1:91,2] = PR[GP1:90,2] + -32.977;
   1:L PR[91] R[100]mm/sec CNT100;
   1:  PR[GP1:91,1] = PR[GP1:90,1] + -5.225;
   1:  PR[GP1:91,2] = PR[GP1:90,2] + -32.128;
   1:L PR[91] R[100]mm/sec CNT100;
   1:  PR[GP1:91,1] = PR[GP1:90,1] + -2.742;
   1:  PR[GP1:91,2] = PR[GP1:90,2] + -30.324;
   1:L PR[91] R[100]mm/sec CNT100;
   1:  PR[GP1:91,1] = PR[GP1:90,1] + -1.241;
   1:  PR[GP1:91,2] = PR[GP1:90,2] + -30.264;
   1:L PR[91] R[100]mm/sec CNT100;
   1:  PR[GP1:91,1] = PR[GP1:90,1] + 1.724;
   1:  PR[GP1:91,2] = PR[GP1:90,2] + -29.631;
   1:L PR[91] R[100]mm/sec CNT100;
   1:  PR[GP1:91,1] = PR[GP1:90,1] + 2.075;
   1:  PR[GP1:91,2] = PR[GP1:90,2] + -29.914;
   1:L PR[91] R[100]mm/sec CNT100;
   1:  PR[GP1:91,1] = PR[GP1:90,1] + 3.056;
   1:  PR[GP1:91,2] = PR[GP1:90,2] + -30.402;
   1:L PR[91] R[100]mm/sec CNT100;
   1:  PR[GP1:91,1] = PR[GP1:90,1] + 5.438;
   1:  PR[GP1:91,2] = PR[GP1:90,2] + -32.133;
   1:L PR[91] R[100]mm/sec CNT100;
   1:  PR[GP1:91,1] = PR[GP1:90,1] + 7.044;
   1:  PR[GP1:91,2] = PR[GP1:90,2] + -32.971;
   1:L PR[91] R[100]mm/sec CNT100;
   1:  PR[GP1:91,1] = PR[GP1:90,1] + 9.068;
   1:  PR[GP1:91,2] = PR[GP1:90,2] + -33.621;
   1:L PR[91] R[100]mm/sec CNT100;
   1:  PR[GP1:91,1] = PR[GP1:90,1] + 18.239;
   1:  PR[GP1:91,2] = PR[GP1:90,2] + -36.796;
   1:L PR[91] R[100]mm/sec CNT100;
   1:  PR[GP1:91,1] = PR[GP1:90,1] + 20.720;
   1:  PR[GP1:91,2] = PR[GP1:90,2] + -37.123;
   1:L PR[91] R[100]mm/sec CNT100;
   1:  PR[GP1:91,1] = PR[GP1:90,1] + 23.655;
   1:  PR[GP1:91,2] = PR[GP1:90,2] + -37.024;
   1:L PR[91] R[100]mm/sec CNT100;
   1:  PR[GP1:91,1] = PR[GP1:90,1] + 32.049;
   1:  PR[GP1:91,2] = PR[GP1:90,2] + -36.987;
   1:L PR[91] R[100]mm/sec CNT100;
   1:  PR[GP1:91,1] = PR[GP1:90,1] + 35.223;
   1:  PR[GP1:91,2] = PR[GP1:90,2] + -36.304;
   1:L PR[91] R[100]mm/sec CNT100;
   1:  PR[GP1:91,1] = PR[GP1:90,1] + 38.738;
   1:  PR[GP1:91,2] = PR[GP1:90,2] + -34.919;
   1:L PR[91] R[100]mm/sec CNT100;
   1:  PR[GP1:91,1] = PR[GP1:90,1] + 45.129;
   1:  PR[GP1:91,2] = PR[GP1:90,2] + -32.654;
   1:L PR[91] R[100]mm/sec CNT100;
   1:  PR[GP1:91,1] = PR[GP1:90,1] + 48.477;
   1:  PR[GP1:91,2] = PR[GP1:90,2] + -30.579;
   1:L PR[91] R[100]mm/sec CNT100;
   1:  PR[GP1:91,1] = PR[GP1:90,1] + 51.749;
   1:  PR[GP1:91,2] = PR[GP1:90,2] + -27.682;
   1:L PR[91] R[100]mm/sec CNT100;
   1:  PR[GP1:91,1] = PR[GP1:90,1] + 55.828;
   1:  PR[GP1:91,2] = PR[GP1:90,2] + -24.380;
   1:L PR[91] R[100]mm/sec CNT100;
   1:  PR[GP1:91,1] = PR[GP1:90,1] + 58.561;
   1:  PR[GP1:91,2] = PR[GP1:90,2] + -20.832;
   1:L PR[91] R[100]mm/sec CNT100;
   1:  PR[GP1:91,1] = PR[GP1:90,1] + 60.849;
   1:  PR[GP1:91,2] = PR[GP1:90,2] + -16.441;
   1:L PR[91] R[100]mm/sec CNT100;
   1:  PR[GP1:91,1] = PR[GP1:90,1] + 62.970;
   1:  PR[GP1:91,2] = PR[GP1:90,2] + -12.908;
   1:L PR[91] R[100]mm/sec CNT100;
   1:  PR[GP1:91,1] = PR[GP1:90,1] + 64.283;
   1:  PR[GP1:91,2] = PR[GP1:90,2] + -8.513;
   1:L PR[91] R[100]mm/sec CNT100;
   1:  PR[GP1:91,1] = PR[GP1:90,1] + 64.740;
   1:  PR[GP1:91,2] = PR[GP1:90,2] + -3.623;
   1:L PR[91] R[100]mm/sec CNT100;
   1:  PR[GP1:91,1] = PR[GP1:90,1] + 65.399;
   1:  PR[GP1:91,2] = PR[GP1:90,2] + -0.045;
   1:L PR[91] R[100]mm/sec CNT100;
   1:  PR[GP1:91,1] = PR[GP1:90,1] + 64.956;
   1:  PR[GP1:91,2] = PR[GP1:90,2] + 4.756;
   1:L PR[91] R[100]mm/sec CNT100;
   1:  PR[GP1:91,1] = PR[GP1:90,1] + 64.291;
   1:  PR[GP1:91,2] = PR[GP1:90,2] + 8.342;
   1:L PR[91] R[100]mm/sec CNT100;
   1:  PR[GP1:91,1] = PR[GP1:90,1] + 62.965;
   1:  PR[GP1:91,2] = PR[GP1:90,2] + 12.781;
   1:L PR[91] R[100]mm/sec CNT100;
   1:  PR[GP1:91,1] = PR[GP1:90,1] + 60.808;
   1:  PR[GP1:91,2] = PR[GP1:90,2] + 16.960;
   1:L PR[91] R[100]mm/sec CNT100;
   1:  PR[GP1:91,1] = PR[GP1:90,1] + 58.574;
   1:  PR[GP1:91,2] = PR[GP1:90,2] + 20.671;
   1:L PR[91] R[100]mm/sec CNT100;
   1:  PR[GP1:91,1] = PR[GP1:90,1] + 55.821;
   1:  PR[GP1:91,2] = PR[GP1:90,2] + 24.246;
   1:L PR[91] R[100]mm/sec CNT100;
   1:  PR[GP1:91,1] = PR[GP1:90,1] + 52.774;
   1:  PR[GP1:91,2] = PR[GP1:90,2] + 26.970;
   1:L PR[91] R[100]mm/sec CNT100;
   1:  PR[GP1:91,1] = PR[GP1:90,1] + 48.493;
   1:  PR[GP1:91,2] = PR[GP1:90,2] + 30.425;
   1:L PR[91] R[100]mm/sec CNT100;
   1:  PR[GP1:91,1] = PR[GP1:90,1] + 45.124;
   1:  PR[GP1:91,2] = PR[GP1:90,2] + 32.514;
   1:L PR[91] R[100]mm/sec CNT100;
   1:  PR[GP1:91,1] = PR[GP1:90,1] + 41.802;
   1:  PR[GP1:91,2] = PR[GP1:90,2] + 33.840;
   1:L PR[91] R[100]mm/sec CNT100;
   1:  PR[GP1:91,1] = PR[GP1:90,1] + 35.243;
   1:  PR[GP1:91,2] = PR[GP1:90,2] + 36.156;
   1:L PR[91] R[100]mm/sec CNT100;
   1:  PR[GP1:91,1] = PR[GP1:90,1] + 32.049;
   1:  PR[GP1:91,2] = PR[GP1:90,2] + 36.844;
   1:L PR[91] R[100]mm/sec CNT100;
   1:  PR[GP1:91,1] = PR[GP1:90,1] + 29.159;
   1:  PR[GP1:91,2] = PR[GP1:90,2] + 36.953;
   1:L PR[91] R[100]mm/sec CNT100;
   1:  PR[GP1:91,1] = PR[GP1:90,1] + 20.743;
   1:  PR[GP1:91,2] = PR[GP1:90,2] + 36.982;
   1:L PR[91] R[100]mm/sec CNT100;
   1:  PR[GP1:91,1] = PR[GP1:90,1] + 18.246;
   1:  PR[GP1:91,2] = PR[GP1:90,2] + 36.654;
   1:L PR[91] R[100]mm/sec CNT100;
   1:  PR[GP1:91,1] = PR[GP1:90,1] + 16.093;
   1:  PR[GP1:91,2] = PR[GP1:90,2] + 35.969;
   1:L PR[91] R[100]mm/sec CNT100;
   1:  PR[GP1:91,1] = PR[GP1:90,1] + 7.065;
   1:  PR[GP1:91,2] = PR[GP1:90,2] + 32.839;
   1:L PR[91] R[100]mm/sec CNT100;
   1:  PR[GP1:91,1] = PR[GP1:90,1] + 5.443;
   1:  PR[GP1:91,2] = PR[GP1:90,2] + 31.992;
   1:L PR[91] R[100]mm/sec CNT100;
   1:  PR[GP1:91,1] = PR[GP1:90,1] + 3.358;
   1:  PR[GP1:91,2] = PR[GP1:90,2] + 30.519;
   1:L PR[91] R[100]mm/sec CNT100;
   1:  PR[GP1:91,1] = PR[GP1:90,1] + 3.362;
   1:  PR[GP1:91,2] = PR[GP1:90,2] + 30.444;
   1:L PR[91] R[100]mm/sec CNT100;
   1:  PR[GP1:91,1] = PR[GP1:90,1] + 1.700;
   1:  PR[GP1:91,2] = PR[GP1:90,2] + 29.518;
   1:L PR[91] R[100]mm/sec CNT100;
   1:  ! -- Layer/Ebene 101 -- !;
   1:  PR[91] = PR[90];
   1:  PR[GP1:91,1] = PR[GP1:90,1] + -0.452;
   1:  PR[GP1:91,2] = PR[GP1:90,2] + 29.941;
   1:  PR[GP1:91,3] = PR[GP1:90,3] + 61.915;
   1:L PR[91] R[100]mm/sec CNT100;
   1:  PR[GP1:91,1] = PR[GP1:90,1] + -2.757;
   1:  PR[GP1:91,2] = PR[GP1:90,2] + 30.477;
   1:L PR[91] R[100]mm/sec CNT100;
   1:  PR[GP1:91,1] = PR[GP1:90,1] + -5.020;
   1:  PR[GP1:91,2] = PR[GP1:90,2] + 32.075;
   1:L PR[91] R[100]mm/sec CNT100;
   1:  PR[GP1:91,1] = PR[GP1:90,1] + -6.515;
   1:  PR[GP1:91,2] = PR[GP1:90,2] + 32.857;
   1:L PR[91] R[100]mm/sec CNT100;
   1:  PR[GP1:91,1] = PR[GP1:90,1] + -8.384;
   1:  PR[GP1:91,2] = PR[GP1:90,2] + 33.458;
   1:L PR[91] R[100]mm/sec CNT100;
   1:  PR[GP1:91,1] = PR[GP1:90,1] + -17.846;
   1:  PR[GP1:91,2] = PR[GP1:90,2] + 36.729;
   1:L PR[91] R[100]mm/sec CNT100;
   1:  PR[GP1:91,1] = PR[GP1:90,1] + -20.178;
   1:  PR[GP1:91,2] = PR[GP1:90,2] + 37.034;
   1:L PR[91] R[100]mm/sec CNT100;
   1:  PR[GP1:91,1] = PR[GP1:90,1] + -22.951;
   1:  PR[GP1:91,2] = PR[GP1:90,2] + 36.938;
   1:L PR[91] R[100]mm/sec CNT100;
   1:  PR[GP1:91,1] = PR[GP1:90,1] + -31.679;
   1:  PR[GP1:91,2] = PR[GP1:90,2] + 36.895;
   1:L PR[91] R[100]mm/sec CNT100;
   1:  PR[GP1:91,1] = PR[GP1:90,1] + -34.700;
   1:  PR[GP1:91,2] = PR[GP1:90,2] + 36.243;
   1:L PR[91] R[100]mm/sec CNT100;
   1:  PR[GP1:91,1] = PR[GP1:90,1] + -38.040;
   1:  PR[GP1:91,2] = PR[GP1:90,2] + 34.921;
   1:L PR[91] R[100]mm/sec CNT100;
   1:  PR[GP1:91,1] = PR[GP1:90,1] + -44.758;
   1:  PR[GP1:91,2] = PR[GP1:90,2] + 32.535;
   1:L PR[91] R[100]mm/sec CNT100;
   1:  PR[GP1:91,1] = PR[GP1:90,1] + -47.984;
   1:  PR[GP1:91,2] = PR[GP1:90,2] + 30.525;
   1:L PR[91] R[100]mm/sec CNT100;
   1:  PR[GP1:91,1] = PR[GP1:90,1] + -51.140;
   1:  PR[GP1:91,2] = PR[GP1:90,2] + 27.723;
   1:L PR[91] R[100]mm/sec CNT100;
   1:  PR[GP1:91,1] = PR[GP1:90,1] + -55.488;
   1:  PR[GP1:91,2] = PR[GP1:90,2] + 24.204;
   1:L PR[91] R[100]mm/sec CNT100;
   1:  PR[GP1:91,1] = PR[GP1:90,1] + -58.092;
   1:  PR[GP1:91,2] = PR[GP1:90,2] + 20.815;
   1:L PR[91] R[100]mm/sec CNT100;
   1:  PR[GP1:91,1] = PR[GP1:90,1] + -60.290;
   1:  PR[GP1:91,2] = PR[GP1:90,2] + 16.550;
   1:L PR[91] R[100]mm/sec CNT100;
   1:  PR[GP1:91,1] = PR[GP1:90,1] + -62.589;
   1:  PR[GP1:91,2] = PR[GP1:90,2] + 12.710;
   1:L PR[91] R[100]mm/sec CNT100;
   1:  PR[GP1:91,1] = PR[GP1:90,1] + -63.858;
   1:  PR[GP1:91,2] = PR[GP1:90,2] + 8.404;
   1:L PR[91] R[100]mm/sec CNT100;
   1:  PR[GP1:91,1] = PR[GP1:90,1] + -64.279;
   1:  PR[GP1:91,2] = PR[GP1:90,2] + 3.807;
   1:L PR[91] R[100]mm/sec CNT100;
   1:  PR[GP1:91,1] = PR[GP1:90,1] + -64.999;
   1:  PR[GP1:91,2] = PR[GP1:90,2] + -0.100;
   1:L PR[91] R[100]mm/sec CNT100;
   1:  PR[GP1:91,1] = PR[GP1:90,1] + -64.591;
   1:  PR[GP1:91,2] = PR[GP1:90,2] + -4.613;
   1:L PR[91] R[100]mm/sec CNT100;
   1:  PR[GP1:91,1] = PR[GP1:90,1] + -63.866;
   1:  PR[GP1:91,2] = PR[GP1:90,2] + -8.523;
   1:L PR[91] R[100]mm/sec CNT100;
   1:  PR[GP1:91,1] = PR[GP1:90,1] + -62.583;
   1:  PR[GP1:91,2] = PR[GP1:90,2] + -12.875;
   1:L PR[91] R[100]mm/sec CNT100;
   1:  PR[GP1:91,1] = PR[GP1:90,1] + -60.507;
   1:  PR[GP1:91,2] = PR[GP1:90,2] + -16.944;
   1:L PR[91] R[100]mm/sec CNT100;
   1:  PR[GP1:91,1] = PR[GP1:90,1] + -58.102;
   1:  PR[GP1:91,2] = PR[GP1:90,2] + -20.946;
   1:L PR[91] R[100]mm/sec CNT100;
   1:  PR[GP1:91,1] = PR[GP1:90,1] + -55.477;
   1:  PR[GP1:91,2] = PR[GP1:90,2] + -24.363;
   1:L PR[91] R[100]mm/sec CNT100;
   1:  PR[GP1:91,1] = PR[GP1:90,1] + -52.527;
   1:  PR[GP1:91,2] = PR[GP1:90,2] + -27.009;
   1:L PR[91] R[100]mm/sec CNT100;
   1:  PR[GP1:91,1] = PR[GP1:90,1] + -47.991;
   1:  PR[GP1:91,2] = PR[GP1:90,2] + -30.664;
   1:L PR[91] R[100]mm/sec CNT100;
   1:  PR[GP1:91,1] = PR[GP1:90,1] + -44.742;
   1:  PR[GP1:91,2] = PR[GP1:90,2] + -32.689;
   1:L PR[91] R[100]mm/sec CNT100;
   1:  PR[GP1:91,1] = PR[GP1:90,1] + -41.562;
   1:  PR[GP1:91,2] = PR[GP1:90,2] + -33.966;
   1:L PR[91] R[100]mm/sec CNT100;
   1:  PR[GP1:91,1] = PR[GP1:90,1] + -34.701;
   1:  PR[GP1:91,2] = PR[GP1:90,2] + -36.386;
   1:L PR[91] R[100]mm/sec CNT100;
   1:  PR[GP1:91,1] = PR[GP1:90,1] + -31.659;
   1:  PR[GP1:91,2] = PR[GP1:90,2] + -37.043;
   1:L PR[91] R[100]mm/sec CNT100;
   1:  PR[GP1:91,1] = PR[GP1:90,1] + -28.898;
   1:  PR[GP1:91,2] = PR[GP1:90,2] + -37.149;
   1:L PR[91] R[100]mm/sec CNT100;
   1:  PR[GP1:91,1] = PR[GP1:90,1] + -20.172;
   1:  PR[GP1:91,2] = PR[GP1:90,2] + -37.177;
   1:L PR[91] R[100]mm/sec CNT100;
   1:  PR[GP1:91,1] = PR[GP1:90,1] + -17.824;
   1:  PR[GP1:91,2] = PR[GP1:90,2] + -36.870;
   1:L PR[91] R[100]mm/sec CNT100;
   1:  PR[GP1:91,1] = PR[GP1:90,1] + -15.804;
   1:  PR[GP1:91,2] = PR[GP1:90,2] + -36.227;
   1:L PR[91] R[100]mm/sec CNT100;
   1:  PR[GP1:91,1] = PR[GP1:90,1] + -6.506;
   1:  PR[GP1:91,2] = PR[GP1:90,2] + -32.996;
   1:L PR[91] R[100]mm/sec CNT100;
   1:  PR[GP1:91,1] = PR[GP1:90,1] + -5.014;
   1:  PR[GP1:91,2] = PR[GP1:90,2] + -32.215;
   1:L PR[91] R[100]mm/sec CNT100;
   1:  PR[GP1:91,1] = PR[GP1:90,1] + -2.714;
   1:  PR[GP1:91,2] = PR[GP1:90,2] + -30.544;
   1:L PR[91] R[100]mm/sec CNT100;
   1:  PR[GP1:91,1] = PR[GP1:90,1] + -1.075;
   1:  PR[GP1:91,2] = PR[GP1:90,2] + -30.479;
   1:L PR[91] R[100]mm/sec CNT100;
   1:  PR[GP1:91,1] = PR[GP1:90,1] + 1.755;
   1:  PR[GP1:91,2] = PR[GP1:90,2] + -29.875;
   1:L PR[91] R[100]mm/sec CNT100;
   1:  PR[GP1:91,1] = PR[GP1:90,1] + 2.124;
   1:  PR[GP1:91,2] = PR[GP1:90,2] + -30.172;
   1:L PR[91] R[100]mm/sec CNT100;
   1:  PR[GP1:91,1] = PR[GP1:90,1] + 3.028;
   1:  PR[GP1:91,2] = PR[GP1:90,2] + -30.622;
   1:L PR[91] R[100]mm/sec CNT100;
   1:  PR[GP1:91,1] = PR[GP1:90,1] + 5.226;
   1:  PR[GP1:91,2] = PR[GP1:90,2] + -32.220;
   1:L PR[91] R[100]mm/sec CNT100;
   1:  PR[GP1:91,1] = PR[GP1:90,1] + 6.702;
   1:  PR[GP1:91,2] = PR[GP1:90,2] + -32.989;
   1:L PR[91] R[100]mm/sec CNT100;
   1:  PR[GP1:91,1] = PR[GP1:90,1] + 8.567;
   1:  PR[GP1:91,2] = PR[GP1:90,2] + -33.589;
   1:L PR[91] R[100]mm/sec CNT100;
   1:  PR[GP1:91,1] = PR[GP1:90,1] + 18.041;
   1:  PR[GP1:91,2] = PR[GP1:90,2] + -36.869;
   1:L PR[91] R[100]mm/sec CNT100;
   1:  PR[GP1:91,1] = PR[GP1:90,1] + 20.368;
   1:  PR[GP1:91,2] = PR[GP1:90,2] + -37.175;
   1:L PR[91] R[100]mm/sec CNT100;
   1:  PR[GP1:91,1] = PR[GP1:90,1] + 23.128;
   1:  PR[GP1:91,2] = PR[GP1:90,2] + -37.082;
   1:L PR[91] R[100]mm/sec CNT100;
   1:  PR[GP1:91,1] = PR[GP1:90,1] + 31.862;
   1:  PR[GP1:91,2] = PR[GP1:90,2] + -37.044;
   1:L PR[91] R[100]mm/sec CNT100;
   1:  PR[GP1:91,1] = PR[GP1:90,1] + 34.878;
   1:  PR[GP1:91,2] = PR[GP1:90,2] + -36.394;
   1:L PR[91] R[100]mm/sec CNT100;
   1:  PR[GP1:91,1] = PR[GP1:90,1] + 38.223;
   1:  PR[GP1:91,2] = PR[GP1:90,2] + -35.077;
   1:L PR[91] R[100]mm/sec CNT100;
   1:  PR[GP1:91,1] = PR[GP1:90,1] + 44.946;
   1:  PR[GP1:91,2] = PR[GP1:90,2] + -32.694;
   1:L PR[91] R[100]mm/sec CNT100;
   1:  PR[GP1:91,1] = PR[GP1:90,1] + 48.153;
   1:  PR[GP1:91,2] = PR[GP1:90,2] + -30.706;
   1:L PR[91] R[100]mm/sec CNT100;
   1:  PR[GP1:91,1] = PR[GP1:90,1] + 51.291;
   1:  PR[GP1:91,2] = PR[GP1:90,2] + -27.928;
   1:L PR[91] R[100]mm/sec CNT100;
   1:  PR[GP1:91,1] = PR[GP1:90,1] + 55.646;
   1:  PR[GP1:91,2] = PR[GP1:90,2] + -24.402;
   1:L PR[91] R[100]mm/sec CNT100;
   1:  PR[GP1:91,1] = PR[GP1:90,1] + 58.277;
   1:  PR[GP1:91,2] = PR[GP1:90,2] + -20.987;
   1:L PR[91] R[100]mm/sec CNT100;
   1:  PR[GP1:91,1] = PR[GP1:90,1] + 60.481;
   1:  PR[GP1:91,2] = PR[GP1:90,2] + -16.757;
   1:L PR[91] R[100]mm/sec CNT100;
   1:  PR[GP1:91,1] = PR[GP1:90,1] + 62.783;
   1:  PR[GP1:91,2] = PR[GP1:90,2] + -12.922;
   1:L PR[91] R[100]mm/sec CNT100;
   1:  PR[GP1:91,1] = PR[GP1:90,1] + 64.050;
   1:  PR[GP1:91,2] = PR[GP1:90,2] + -8.680;
   1:L PR[91] R[100]mm/sec CNT100;
   1:  PR[GP1:91,1] = PR[GP1:90,1] + 64.492;
   1:  PR[GP1:91,2] = PR[GP1:90,2] + -3.957;
   1:L PR[91] R[100]mm/sec CNT100;
   1:  PR[GP1:91,1] = PR[GP1:90,1] + 65.212;
   1:  PR[GP1:91,2] = PR[GP1:90,2] + -0.045;
   1:L PR[91] R[100]mm/sec CNT100;
   1:  PR[GP1:91,1] = PR[GP1:90,1] + 64.784;
   1:  PR[GP1:91,2] = PR[GP1:90,2] + 4.595;
   1:L PR[91] R[100]mm/sec CNT100;
   1:  PR[GP1:91,1] = PR[GP1:90,1] + 64.059;
   1:  PR[GP1:91,2] = PR[GP1:90,2] + 8.509;
   1:L PR[91] R[100]mm/sec CNT100;
   1:  PR[GP1:91,1] = PR[GP1:90,1] + 62.778;
   1:  PR[GP1:91,2] = PR[GP1:90,2] + 12.795;
   1:L PR[91] R[100]mm/sec CNT100;
   1:  PR[GP1:91,1] = PR[GP1:90,1] + 60.696;
   1:  PR[GP1:91,2] = PR[GP1:90,2] + 16.830;
   1:L PR[91] R[100]mm/sec CNT100;
   1:  PR[GP1:91,1] = PR[GP1:90,1] + 58.290;
   1:  PR[GP1:91,2] = PR[GP1:90,2] + 20.826;
   1:L PR[91] R[100]mm/sec CNT100;
   1:  PR[GP1:91,1] = PR[GP1:90,1] + 55.639;
   1:  PR[GP1:91,2] = PR[GP1:90,2] + 24.268;
   1:L PR[91] R[100]mm/sec CNT100;
   1:  PR[GP1:91,1] = PR[GP1:90,1] + 52.705;
   1:  PR[GP1:91,2] = PR[GP1:90,2] + 26.891;
   1:L PR[91] R[100]mm/sec CNT100;
   1:  PR[GP1:91,1] = PR[GP1:90,1] + 48.170;
   1:  PR[GP1:91,2] = PR[GP1:90,2] + 30.552;
   1:L PR[91] R[100]mm/sec CNT100;
   1:  PR[GP1:91,1] = PR[GP1:90,1] + 44.942;
   1:  PR[GP1:91,2] = PR[GP1:90,2] + 32.553;
   1:L PR[91] R[100]mm/sec CNT100;
   1:  PR[GP1:91,1] = PR[GP1:90,1] + 41.758;
   1:  PR[GP1:91,2] = PR[GP1:90,2] + 33.825;
   1:L PR[91] R[100]mm/sec CNT100;
   1:  PR[GP1:91,1] = PR[GP1:90,1] + 34.899;
   1:  PR[GP1:91,2] = PR[GP1:90,2] + 36.246;
   1:L PR[91] R[100]mm/sec CNT100;
   1:  PR[GP1:91,1] = PR[GP1:90,1] + 31.862;
   1:  PR[GP1:91,2] = PR[GP1:90,2] + 36.900;
   1:L PR[91] R[100]mm/sec CNT100;
   1:  PR[GP1:91,1] = PR[GP1:90,1] + 29.114;
   1:  PR[GP1:91,2] = PR[GP1:90,2] + 37.004;
   1:L PR[91] R[100]mm/sec CNT100;
   1:  PR[GP1:91,1] = PR[GP1:90,1] + 20.392;
   1:  PR[GP1:91,2] = PR[GP1:90,2] + 37.034;
   1:L PR[91] R[100]mm/sec CNT100;
   1:  PR[GP1:91,1] = PR[GP1:90,1] + 18.047;
   1:  PR[GP1:91,2] = PR[GP1:90,2] + 36.726;
   1:L PR[91] R[100]mm/sec CNT100;
   1:  PR[GP1:91,1] = PR[GP1:90,1] + 16.025;
   1:  PR[GP1:91,2] = PR[GP1:90,2] + 36.083;
   1:L PR[91] R[100]mm/sec CNT100;
   1:  PR[GP1:91,1] = PR[GP1:90,1] + 6.723;
   1:  PR[GP1:91,2] = PR[GP1:90,2] + 32.858;
   1:L PR[91] R[100]mm/sec CNT100;
   1:  PR[GP1:91,1] = PR[GP1:90,1] + 5.232;
   1:  PR[GP1:91,2] = PR[GP1:90,2] + 32.079;
   1:L PR[91] R[100]mm/sec CNT100;
   1:  PR[GP1:91,1] = PR[GP1:90,1] + 3.330;
   1:  PR[GP1:91,2] = PR[GP1:90,2] + 30.736;
   1:L PR[91] R[100]mm/sec CNT100;
   1:  PR[GP1:91,1] = PR[GP1:90,1] + 3.334;
   1:  PR[GP1:91,2] = PR[GP1:90,2] + 30.655;
   1:L PR[91] R[100]mm/sec CNT100;
   1:  PR[GP1:91,1] = PR[GP1:90,1] + 1.730;
   1:  PR[GP1:91,2] = PR[GP1:90,2] + 29.762;
   1:L PR[91] R[100]mm/sec CNT100;
   1:  ! -- Layer/Ebene 102 -- !;
   1:  PR[91] = PR[90];
   1:  PR[GP1:91,1] = PR[GP1:90,1] + -0.603;
   1:  PR[GP1:91,2] = PR[GP1:90,2] + 30.199;
   1:  PR[GP1:91,3] = PR[GP1:90,3] + 62.525;
   1:L PR[91] R[100]mm/sec CNT100;
   1:  PR[GP1:91,1] = PR[GP1:90,1] + -2.730;
   1:  PR[GP1:91,2] = PR[GP1:90,2] + 30.693;
   1:L PR[91] R[100]mm/sec CNT100;
   1:  PR[GP1:91,1] = PR[GP1:90,1] + -4.809;
   1:  PR[GP1:91,2] = PR[GP1:90,2] + 32.163;
   1:L PR[91] R[100]mm/sec CNT100;
   1:  PR[GP1:91,1] = PR[GP1:90,1] + -6.173;
   1:  PR[GP1:91,2] = PR[GP1:90,2] + 32.876;
   1:L PR[91] R[100]mm/sec CNT100;
   1:  PR[GP1:91,1] = PR[GP1:90,1] + -7.884;
   1:  PR[GP1:91,2] = PR[GP1:90,2] + 33.426;
   1:L PR[91] R[100]mm/sec CNT100;
   1:  PR[GP1:91,1] = PR[GP1:90,1] + -17.648;
   1:  PR[GP1:91,2] = PR[GP1:90,2] + 36.801;
   1:L PR[91] R[100]mm/sec CNT100;
   1:  PR[GP1:91,1] = PR[GP1:90,1] + -19.826;
   1:  PR[GP1:91,2] = PR[GP1:90,2] + 37.086;
   1:L PR[91] R[100]mm/sec CNT100;
   1:  PR[GP1:91,1] = PR[GP1:90,1] + -22.422;
   1:  PR[GP1:91,2] = PR[GP1:90,2] + 36.997;
   1:L PR[91] R[100]mm/sec CNT100;
   1:  PR[GP1:91,1] = PR[GP1:90,1] + -31.491;
   1:  PR[GP1:91,2] = PR[GP1:90,2] + 36.951;
   1:L PR[91] R[100]mm/sec CNT100;
   1:  PR[GP1:91,1] = PR[GP1:90,1] + -34.354;
   1:  PR[GP1:91,2] = PR[GP1:90,2] + 36.334;
   1:L PR[91] R[100]mm/sec CNT100;
   1:  PR[GP1:91,1] = PR[GP1:90,1] + -37.524;
   1:  PR[GP1:91,2] = PR[GP1:90,2] + 35.079;
   1:L PR[91] R[100]mm/sec CNT100;
   1:  PR[GP1:91,1] = PR[GP1:90,1] + -44.574;
   1:  PR[GP1:91,2] = PR[GP1:90,2] + 32.575;
   1:L PR[91] R[100]mm/sec CNT100;
   1:  PR[GP1:91,1] = PR[GP1:90,1] + -47.660;
   1:  PR[GP1:91,2] = PR[GP1:90,2] + 30.653;
   1:L PR[91] R[100]mm/sec CNT100;
   1:  PR[GP1:91,1] = PR[GP1:90,1] + -50.679;
   1:  PR[GP1:91,2] = PR[GP1:90,2] + 27.972;
   1:L PR[91] R[100]mm/sec CNT100;
   1:  PR[GP1:91,1] = PR[GP1:90,1] + -55.305;
   1:  PR[GP1:91,2] = PR[GP1:90,2] + 24.228;
   1:L PR[91] R[100]mm/sec CNT100;
   1:  PR[GP1:91,1] = PR[GP1:90,1] + -57.808;
   1:  PR[GP1:91,2] = PR[GP1:90,2] + 20.971;
   1:L PR[91] R[100]mm/sec CNT100;
   1:  PR[GP1:91,1] = PR[GP1:90,1] + -59.922;
   1:  PR[GP1:91,2] = PR[GP1:90,2] + 16.868;
   1:L PR[91] R[100]mm/sec CNT100;
   1:  PR[GP1:91,1] = PR[GP1:90,1] + -62.402;
   1:  PR[GP1:91,2] = PR[GP1:90,2] + 12.725;
   1:L PR[91] R[100]mm/sec CNT100;
   1:  PR[GP1:91,1] = PR[GP1:90,1] + -63.625;
   1:  PR[GP1:91,2] = PR[GP1:90,2] + 8.576;
   1:L PR[91] R[100]mm/sec CNT100;
   1:  PR[GP1:91,1] = PR[GP1:90,1] + -64.031;
   1:  PR[GP1:91,2] = PR[GP1:90,2] + 4.142;
   1:L PR[91] R[100]mm/sec CNT100;
   1:  PR[GP1:91,1] = PR[GP1:90,1] + -64.813;
   1:  PR[GP1:91,2] = PR[GP1:90,2] + -0.100;
   1:L PR[91] R[100]mm/sec CNT100;
   1:  PR[GP1:91,1] = PR[GP1:90,1] + -64.419;
   1:  PR[GP1:91,2] = PR[GP1:90,2] + -4.457;
   1:L PR[91] R[100]mm/sec CNT100;
   1:  PR[GP1:91,1] = PR[GP1:90,1] + -63.633;
   1:  PR[GP1:91,2] = PR[GP1:90,2] + -8.694;
   1:L PR[91] R[100]mm/sec CNT100;
   1:  PR[GP1:91,1] = PR[GP1:90,1] + -62.396;
   1:  PR[GP1:91,2] = PR[GP1:90,2] + -12.890;
   1:L PR[91] R[100]mm/sec CNT100;
   1:  PR[GP1:91,1] = PR[GP1:90,1] + -60.395;
   1:  PR[GP1:91,2] = PR[GP1:90,2] + -16.814;
   1:L PR[91] R[100]mm/sec CNT100;
   1:  PR[GP1:91,1] = PR[GP1:90,1] + -57.817;
   1:  PR[GP1:91,2] = PR[GP1:90,2] + -21.102;
   1:L PR[91] R[100]mm/sec CNT100;
   1:  PR[GP1:91,1] = PR[GP1:90,1] + -55.293;
   1:  PR[GP1:91,2] = PR[GP1:90,2] + -24.387;
   1:L PR[91] R[100]mm/sec CNT100;
   1:  PR[GP1:91,1] = PR[GP1:90,1] + -52.457;
   1:  PR[GP1:91,2] = PR[GP1:90,2] + -26.931;
   1:L PR[91] R[100]mm/sec CNT100;
   1:  PR[GP1:91,1] = PR[GP1:90,1] + -47.666;
   1:  PR[GP1:91,2] = PR[GP1:90,2] + -30.793;
   1:L PR[91] R[100]mm/sec CNT100;
   1:  PR[GP1:91,1] = PR[GP1:90,1] + -44.558;
   1:  PR[GP1:91,2] = PR[GP1:90,2] + -32.729;
   1:L PR[91] R[100]mm/sec CNT100;
   1:  PR[GP1:91,1] = PR[GP1:90,1] + -41.516;
   1:  PR[GP1:91,2] = PR[GP1:90,2] + -33.950;
   1:L PR[91] R[100]mm/sec CNT100;
   1:  PR[GP1:91,1] = PR[GP1:90,1] + -34.355;
   1:  PR[GP1:91,2] = PR[GP1:90,2] + -36.477;
   1:L PR[91] R[100]mm/sec CNT100;
   1:  PR[GP1:91,1] = PR[GP1:90,1] + -31.471;
   1:  PR[GP1:91,2] = PR[GP1:90,2] + -37.099;
   1:L PR[91] R[100]mm/sec CNT100;
   1:  PR[GP1:91,1] = PR[GP1:90,1] + -28.852;
   1:  PR[GP1:91,2] = PR[GP1:90,2] + -37.200;
   1:L PR[91] R[100]mm/sec CNT100;
   1:  PR[GP1:91,1] = PR[GP1:90,1] + -19.820;
   1:  PR[GP1:91,2] = PR[GP1:90,2] + -37.229;
   1:L PR[91] R[100]mm/sec CNT100;
   1:  PR[GP1:91,1] = PR[GP1:90,1] + -17.625;
   1:  PR[GP1:91,2] = PR[GP1:90,2] + -36.942;
   1:L PR[91] R[100]mm/sec CNT100;
   1:  PR[GP1:91,1] = PR[GP1:90,1] + -15.736;
   1:  PR[GP1:91,2] = PR[GP1:90,2] + -36.341;
   1:L PR[91] R[100]mm/sec CNT100;
   1:  PR[GP1:91,1] = PR[GP1:90,1] + -6.163;
   1:  PR[GP1:91,2] = PR[GP1:90,2] + -33.014;
   1:L PR[91] R[100]mm/sec CNT100;
   1:  PR[GP1:91,1] = PR[GP1:90,1] + -4.803;
   1:  PR[GP1:91,2] = PR[GP1:90,2] + -32.303;
   1:L PR[91] R[100]mm/sec CNT100;
   1:  PR[GP1:91,1] = PR[GP1:90,1] + -2.686;
   1:  PR[GP1:91,2] = PR[GP1:90,2] + -30.765;
   1:L PR[91] R[100]mm/sec CNT100;
   1:  PR[GP1:91,1] = PR[GP1:90,1] + -0.910;
   1:  PR[GP1:91,2] = PR[GP1:90,2] + -30.694;
   1:L PR[91] R[100]mm/sec CNT100;
   1:  PR[GP1:91,1] = PR[GP1:90,1] + 1.785;
   1:  PR[GP1:91,2] = PR[GP1:90,2] + -30.119;
   1:L PR[91] R[100]mm/sec CNT100;
   1:  PR[GP1:91,1] = PR[GP1:90,1] + 2.173;
   1:  PR[GP1:91,2] = PR[GP1:90,2] + -30.431;
   1:L PR[91] R[100]mm/sec CNT100;
   1:  PR[GP1:91,1] = PR[GP1:90,1] + 3.000;
   1:  PR[GP1:91,2] = PR[GP1:90,2] + -30.842;
   1:L PR[91] R[100]mm/sec CNT100;
   1:  PR[GP1:91,1] = PR[GP1:90,1] + 5.015;
   1:  PR[GP1:91,2] = PR[GP1:90,2] + -32.306;
   1:L PR[91] R[100]mm/sec CNT100;
   1:  PR[GP1:91,1] = PR[GP1:90,1] + 6.360;
   1:  PR[GP1:91,2] = PR[GP1:90,2] + -33.008;
   1:L PR[91] R[100]mm/sec CNT100;
   1:  PR[GP1:91,1] = PR[GP1:90,1] + 8.065;
   1:  PR[GP1:91,2] = PR[GP1:90,2] + -33.556;
   1:L PR[91] R[100]mm/sec CNT100;
   1:  PR[GP1:91,1] = PR[GP1:90,1] + 17.842;
   1:  PR[GP1:91,2] = PR[GP1:90,2] + -36.941;
   1:L PR[91] R[100]mm/sec CNT100;
   1:  PR[GP1:91,1] = PR[GP1:90,1] + 20.017;
   1:  PR[GP1:91,2] = PR[GP1:90,2] + -37.227;
   1:L PR[91] R[100]mm/sec CNT100;
   1:  PR[GP1:91,1] = PR[GP1:90,1] + 22.600;
   1:  PR[GP1:91,2] = PR[GP1:90,2] + -37.140;
   1:L PR[91] R[100]mm/sec CNT100;
   1:  PR[GP1:91,1] = PR[GP1:90,1] + 31.675;
   1:  PR[GP1:91,2] = PR[GP1:90,2] + -37.100;
   1:L PR[91] R[100]mm/sec CNT100;
   1:  PR[GP1:91,1] = PR[GP1:90,1] + 34.533;
   1:  PR[GP1:91,2] = PR[GP1:90,2] + -36.485;
   1:L PR[91] R[100]mm/sec CNT100;
   1:  PR[GP1:91,1] = PR[GP1:90,1] + 37.707;
   1:  PR[GP1:91,2] = PR[GP1:90,2] + -35.235;
   1:L PR[91] R[100]mm/sec CNT100;
   1:  PR[GP1:91,1] = PR[GP1:90,1] + 44.763;
   1:  PR[GP1:91,2] = PR[GP1:90,2] + -32.734;
   1:L PR[91] R[100]mm/sec CNT100;
   1:  PR[GP1:91,1] = PR[GP1:90,1] + 47.829;
   1:  PR[GP1:91,2] = PR[GP1:90,2] + -30.833;
   1:L PR[91] R[100]mm/sec CNT100;
   1:  PR[GP1:91,1] = PR[GP1:90,1] + 50.832;
   1:  PR[GP1:91,2] = PR[GP1:90,2] + -28.174;
   1:L PR[91] R[100]mm/sec CNT100;
   1:  PR[GP1:91,1] = PR[GP1:90,1] + 55.465;
   1:  PR[GP1:91,2] = PR[GP1:90,2] + -24.425;
   1:L PR[91] R[100]mm/sec CNT100;
   1:  PR[GP1:91,1] = PR[GP1:90,1] + 57.993;
   1:  PR[GP1:91,2] = PR[GP1:90,2] + -21.142;
   1:L PR[91] R[100]mm/sec CNT100;
   1:  PR[GP1:91,1] = PR[GP1:90,1] + 60.114;
   1:  PR[GP1:91,2] = PR[GP1:90,2] + -17.073;
   1:L PR[91] R[100]mm/sec CNT100;
   1:  PR[GP1:91,1] = PR[GP1:90,1] + 62.597;
   1:  PR[GP1:91,2] = PR[GP1:90,2] + -12.936;
   1:L PR[91] R[100]mm/sec CNT100;
   1:  PR[GP1:91,1] = PR[GP1:90,1] + 63.818;
   1:  PR[GP1:91,2] = PR[GP1:90,2] + -8.848;
   1:L PR[91] R[100]mm/sec CNT100;
   1:  PR[GP1:91,1] = PR[GP1:90,1] + 64.244;
   1:  PR[GP1:91,2] = PR[GP1:90,2] + -4.292;
   1:L PR[91] R[100]mm/sec CNT100;
   1:  PR[GP1:91,1] = PR[GP1:90,1] + 65.026;
   1:  PR[GP1:91,2] = PR[GP1:90,2] + -0.045;
   1:L PR[91] R[100]mm/sec CNT100;
   1:  PR[GP1:91,1] = PR[GP1:90,1] + 64.613;
   1:  PR[GP1:91,2] = PR[GP1:90,2] + 4.434;
   1:L PR[91] R[100]mm/sec CNT100;
   1:  PR[GP1:91,1] = PR[GP1:90,1] + 63.826;
   1:  PR[GP1:91,2] = PR[GP1:90,2] + 8.677;
   1:L PR[91] R[100]mm/sec CNT100;
   1:  PR[GP1:91,1] = PR[GP1:90,1] + 62.592;
   1:  PR[GP1:91,2] = PR[GP1:90,2] + 12.809;
   1:L PR[91] R[100]mm/sec CNT100;
   1:  PR[GP1:91,1] = PR[GP1:90,1] + 60.584;
   1:  PR[GP1:91,2] = PR[GP1:90,2] + 16.699;
   1:L PR[91] R[100]mm/sec CNT100;
   1:  PR[GP1:91,1] = PR[GP1:90,1] + 58.007;
   1:  PR[GP1:91,2] = PR[GP1:90,2] + 20.980;
   1:L PR[91] R[100]mm/sec CNT100;
   1:  PR[GP1:91,1] = PR[GP1:90,1] + 55.458;
   1:  PR[GP1:91,2] = PR[GP1:90,2] + 24.290;
   1:L PR[91] R[100]mm/sec CNT100;
   1:  PR[GP1:91,1] = PR[GP1:90,1] + 52.636;
   1:  PR[GP1:91,2] = PR[GP1:90,2] + 26.812;
   1:L PR[91] R[100]mm/sec CNT100;
   1:  PR[GP1:91,1] = PR[GP1:90,1] + 47.847;
   1:  PR[GP1:91,2] = PR[GP1:90,2] + 30.679;
   1:L PR[91] R[100]mm/sec CNT100;
   1:  PR[GP1:91,1] = PR[GP1:90,1] + 44.759;
   1:  PR[GP1:91,2] = PR[GP1:90,2] + 32.593;
   1:L PR[91] R[100]mm/sec CNT100;
   1:  PR[GP1:91,1] = PR[GP1:90,1] + 41.713;
   1:  PR[GP1:91,2] = PR[GP1:90,2] + 33.809;
   1:L PR[91] R[100]mm/sec CNT100;
   1:  PR[GP1:91,1] = PR[GP1:90,1] + 34.554;
   1:  PR[GP1:91,2] = PR[GP1:90,2] + 36.337;
   1:L PR[91] R[100]mm/sec CNT100;
   1:  PR[GP1:91,1] = PR[GP1:90,1] + 31.675;
   1:  PR[GP1:91,2] = PR[GP1:90,2] + 36.957;
   1:L PR[91] R[100]mm/sec CNT100;
   1:  PR[GP1:91,1] = PR[GP1:90,1] + 29.069;
   1:  PR[GP1:91,2] = PR[GP1:90,2] + 37.055;
   1:L PR[91] R[100]mm/sec CNT100;
   1:  PR[GP1:91,1] = PR[GP1:90,1] + 20.041;
   1:  PR[GP1:91,2] = PR[GP1:90,2] + 37.086;
   1:L PR[91] R[100]mm/sec CNT100;
   1:  PR[GP1:91,1] = PR[GP1:90,1] + 17.849;
   1:  PR[GP1:91,2] = PR[GP1:90,2] + 36.798;
   1:L PR[91] R[100]mm/sec CNT100;
   1:  PR[GP1:91,1] = PR[GP1:90,1] + 15.957;
   1:  PR[GP1:91,2] = PR[GP1:90,2] + 36.196;
   1:L PR[91] R[100]mm/sec CNT100;
   1:  PR[GP1:91,1] = PR[GP1:90,1] + 6.382;
   1:  PR[GP1:91,2] = PR[GP1:90,2] + 32.877;
   1:L PR[91] R[100]mm/sec CNT100;
   1:  PR[GP1:91,1] = PR[GP1:90,1] + 5.021;
   1:  PR[GP1:91,2] = PR[GP1:90,2] + 32.166;
   1:L PR[91] R[100]mm/sec CNT100;
   1:  PR[GP1:91,1] = PR[GP1:90,1] + 3.302;
   1:  PR[GP1:91,2] = PR[GP1:90,2] + 30.952;
   1:L PR[91] R[100]mm/sec CNT100;
   1:  PR[GP1:91,1] = PR[GP1:90,1] + 3.307;
   1:  PR[GP1:91,2] = PR[GP1:90,2] + 30.866;
   1:L PR[91] R[100]mm/sec CNT100;
   1:  PR[GP1:91,1] = PR[GP1:90,1] + 1.760;
   1:  PR[GP1:91,2] = PR[GP1:90,2] + 30.005;
   1:L PR[91] R[100]mm/sec CNT100;
   1:  ! -- Layer/Ebene 103 -- !;
   1:  PR[91] = PR[90];
   1:  PR[GP1:91,1] = PR[GP1:90,1] + -0.754;
   1:  PR[GP1:91,2] = PR[GP1:90,2] + 30.457;
   1:  PR[GP1:91,3] = PR[GP1:90,3] + 63.135;
   1:L PR[91] R[100]mm/sec CNT100;
   1:  PR[GP1:91,1] = PR[GP1:90,1] + -2.702;
   1:  PR[GP1:91,2] = PR[GP1:90,2] + 30.910;
   1:L PR[91] R[100]mm/sec CNT100;
   1:  PR[GP1:91,1] = PR[GP1:90,1] + -4.598;
   1:  PR[GP1:91,2] = PR[GP1:90,2] + 32.250;
   1:L PR[91] R[100]mm/sec CNT100;
   1:  PR[GP1:91,1] = PR[GP1:90,1] + -5.831;
   1:  PR[GP1:91,2] = PR[GP1:90,2] + 32.895;
   1:L PR[91] R[100]mm/sec CNT100;
   1:  PR[GP1:91,1] = PR[GP1:90,1] + -7.383;
   1:  PR[GP1:91,2] = PR[GP1:90,2] + 33.393;
   1:L PR[91] R[100]mm/sec CNT100;
   1:  PR[GP1:91,1] = PR[GP1:90,1] + -17.449;
   1:  PR[GP1:91,2] = PR[GP1:90,2] + 36.874;
   1:L PR[91] R[100]mm/sec CNT100;
   1:  PR[GP1:91,1] = PR[GP1:90,1] + -19.474;
   1:  PR[GP1:91,2] = PR[GP1:90,2] + 37.138;
   1:L PR[91] R[100]mm/sec CNT100;
   1:  PR[GP1:91,1] = PR[GP1:90,1] + -21.894;
   1:  PR[GP1:91,2] = PR[GP1:90,2] + 37.055;
   1:L PR[91] R[100]mm/sec CNT100;
   1:  PR[GP1:91,1] = PR[GP1:90,1] + -31.304;
   1:  PR[GP1:91,2] = PR[GP1:90,2] + 37.008;
   1:L PR[91] R[100]mm/sec CNT100;
   1:  PR[GP1:91,1] = PR[GP1:90,1] + -34.009;
   1:  PR[GP1:91,2] = PR[GP1:90,2] + 36.424;
   1:L PR[91] R[100]mm/sec CNT100;
   1:  PR[GP1:91,1] = PR[GP1:90,1] + -37.008;
   1:  PR[GP1:91,2] = PR[GP1:90,2] + 35.237;
   1:L PR[91] R[100]mm/sec CNT100;
   1:  PR[GP1:91,1] = PR[GP1:90,1] + -44.391;
   1:  PR[GP1:91,2] = PR[GP1:90,2] + 32.615;
   1:L PR[91] R[100]mm/sec CNT100;
   1:  PR[GP1:91,1] = PR[GP1:90,1] + -47.335;
   1:  PR[GP1:91,2] = PR[GP1:90,2] + 30.781;
   1:L PR[91] R[100]mm/sec CNT100;
   1:  PR[GP1:91,1] = PR[GP1:90,1] + -50.219;
   1:  PR[GP1:91,2] = PR[GP1:90,2] + 28.220;
   1:L PR[91] R[100]mm/sec CNT100;
   1:  PR[GP1:91,1] = PR[GP1:90,1] + -55.122;
   1:  PR[GP1:91,2] = PR[GP1:90,2] + 24.253;
   1:L PR[91] R[100]mm/sec CNT100;
   1:  PR[GP1:91,1] = PR[GP1:90,1] + -57.523;
   1:  PR[GP1:91,2] = PR[GP1:90,2] + 21.127;
   1:L PR[91] R[100]mm/sec CNT100;
   1:  PR[GP1:91,1] = PR[GP1:90,1] + -59.554;
   1:  PR[GP1:91,2] = PR[GP1:90,2] + 17.187;
   1:L PR[91] R[100]mm/sec CNT100;
   1:  PR[GP1:91,1] = PR[GP1:90,1] + -62.215;
   1:  PR[GP1:91,2] = PR[GP1:90,2] + 12.741;
   1:L PR[91] R[100]mm/sec CNT100;
   1:  PR[GP1:91,1] = PR[GP1:90,1] + -63.392;
   1:  PR[GP1:91,2] = PR[GP1:90,2] + 8.747;
   1:L PR[91] R[100]mm/sec CNT100;
   1:  PR[GP1:91,1] = PR[GP1:90,1] + -63.783;
   1:  PR[GP1:91,2] = PR[GP1:90,2] + 4.476;
   1:L PR[91] R[100]mm/sec CNT100;
   1:  PR[GP1:91,1] = PR[GP1:90,1] + -64.627;
   1:  PR[GP1:91,2] = PR[GP1:90,2] + -0.100;
   1:L PR[91] R[100]mm/sec CNT100;
   1:  PR[GP1:91,1] = PR[GP1:90,1] + -64.247;
   1:  PR[GP1:91,2] = PR[GP1:90,2] + -4.301;
   1:L PR[91] R[100]mm/sec CNT100;
   1:  PR[GP1:91,1] = PR[GP1:90,1] + -63.400;
   1:  PR[GP1:91,2] = PR[GP1:90,2] + -8.866;
   1:L PR[91] R[100]mm/sec CNT100;
   1:  PR[GP1:91,1] = PR[GP1:90,1] + -62.209;
   1:  PR[GP1:91,2] = PR[GP1:90,2] + -12.906;
   1:L PR[91] R[100]mm/sec CNT100;
   1:  PR[GP1:91,1] = PR[GP1:90,1] + -60.282;
   1:  PR[GP1:91,2] = PR[GP1:90,2] + -16.684;
   1:L PR[91] R[100]mm/sec CNT100;
   1:  PR[GP1:91,1] = PR[GP1:90,1] + -57.533;
   1:  PR[GP1:91,2] = PR[GP1:90,2] + -21.258;
   1:L PR[91] R[100]mm/sec CNT100;
   1:  PR[GP1:91,1] = PR[GP1:90,1] + -55.110;
   1:  PR[GP1:91,2] = PR[GP1:90,2] + -24.412;
   1:L PR[91] R[100]mm/sec CNT100;
   1:  PR[GP1:91,1] = PR[GP1:90,1] + -52.387;
   1:  PR[GP1:91,2] = PR[GP1:90,2] + -26.854;
   1:L PR[91] R[100]mm/sec CNT100;
   1:  PR[GP1:91,1] = PR[GP1:90,1] + -47.341;
   1:  PR[GP1:91,2] = PR[GP1:90,2] + -30.921;
   1:L PR[91] R[100]mm/sec CNT100;
   1:  PR[GP1:91,1] = PR[GP1:90,1] + -44.374;
   1:  PR[GP1:91,2] = PR[GP1:90,2] + -32.769;
   1:L PR[91] R[100]mm/sec CNT100;
   1:  PR[GP1:91,1] = PR[GP1:90,1] + -41.471;
   1:  PR[GP1:91,2] = PR[GP1:90,2] + -33.935;
   1:L PR[91] R[100]mm/sec CNT100;
   1:  PR[GP1:91,1] = PR[GP1:90,1] + -34.009;
   1:  PR[GP1:91,2] = PR[GP1:90,2] + -36.568;
   1:L PR[91] R[100]mm/sec CNT100;
   1:  PR[GP1:91,1] = PR[GP1:90,1] + -31.283;
   1:  PR[GP1:91,2] = PR[GP1:90,2] + -37.156;
   1:L PR[91] R[100]mm/sec CNT100;
   1:  PR[GP1:91,1] = PR[GP1:90,1] + -28.806;
   1:  PR[GP1:91,2] = PR[GP1:90,2] + -37.251;
   1:L PR[91] R[100]mm/sec CNT100;
   1:  PR[GP1:91,1] = PR[GP1:90,1] + -19.468;
   1:  PR[GP1:91,2] = PR[GP1:90,2] + -37.281;
   1:L PR[91] R[100]mm/sec CNT100;
   1:  PR[GP1:91,1] = PR[GP1:90,1] + -17.426;
   1:  PR[GP1:91,2] = PR[GP1:90,2] + -37.014;
   1:L PR[91] R[100]mm/sec CNT100;
   1:  PR[GP1:91,1] = PR[GP1:90,1] + -15.668;
   1:  PR[GP1:91,2] = PR[GP1:90,2] + -36.454;
   1:L PR[91] R[100]mm/sec CNT100;
   1:  PR[GP1:91,1] = PR[GP1:90,1] + -5.821;
   1:  PR[GP1:91,2] = PR[GP1:90,2] + -33.033;
   1:L PR[91] R[100]mm/sec CNT100;
   1:  PR[GP1:91,1] = PR[GP1:90,1] + -4.592;
   1:  PR[GP1:91,2] = PR[GP1:90,2] + -32.390;
   1:L PR[91] R[100]mm/sec CNT100;
   1:  PR[GP1:91,1] = PR[GP1:90,1] + -2.658;
   1:  PR[GP1:91,2] = PR[GP1:90,2] + -30.985;
   1:L PR[91] R[100]mm/sec CNT100;
   1:  PR[GP1:91,1] = PR[GP1:90,1] + -0.744;
   1:  PR[GP1:91,2] = PR[GP1:90,2] + -30.908;
   1:L PR[91] R[100]mm/sec CNT100;
   1:  PR[GP1:91,1] = PR[GP1:90,1] + 1.815;
   1:  PR[GP1:91,2] = PR[GP1:90,2] + -30.362;
   1:L PR[91] R[100]mm/sec CNT100;
   1:  PR[GP1:91,1] = PR[GP1:90,1] + 2.221;
   1:  PR[GP1:91,2] = PR[GP1:90,2] + -30.689;
   1:L PR[91] R[100]mm/sec CNT100;
   1:  PR[GP1:91,1] = PR[GP1:90,1] + 2.972;
   1:  PR[GP1:91,2] = PR[GP1:90,2] + -31.063;
   1:L PR[91] R[100]mm/sec CNT100;
   1:  PR[GP1:91,1] = PR[GP1:90,1] + 4.803;
   1:  PR[GP1:91,2] = PR[GP1:90,2] + -32.393;
   1:L PR[91] R[100]mm/sec CNT100;
   1:  PR[GP1:91,1] = PR[GP1:90,1] + 6.018;
   1:  PR[GP1:91,2] = PR[GP1:90,2] + -33.027;
   1:L PR[91] R[100]mm/sec CNT100;
   1:  PR[GP1:91,1] = PR[GP1:90,1] + 7.563;
   1:  PR[GP1:91,2] = PR[GP1:90,2] + -33.523;
   1:L PR[91] R[100]mm/sec CNT100;
   1:  PR[GP1:91,1] = PR[GP1:90,1] + 17.643;
   1:  PR[GP1:91,2] = PR[GP1:90,2] + -37.013;
   1:L PR[91] R[100]mm/sec CNT100;
   1:  PR[GP1:91,1] = PR[GP1:90,1] + 19.665;
   1:  PR[GP1:91,2] = PR[GP1:90,2] + -37.279;
   1:L PR[91] R[100]mm/sec CNT100;
   1:  PR[GP1:91,1] = PR[GP1:90,1] + 22.072;
   1:  PR[GP1:91,2] = PR[GP1:90,2] + -37.198;
   1:L PR[91] R[100]mm/sec CNT100;
   1:  PR[GP1:91,1] = PR[GP1:90,1] + 31.487;
   1:  PR[GP1:91,2] = PR[GP1:90,2] + -37.157;
   1:L PR[91] R[100]mm/sec CNT100;
   1:  PR[GP1:91,1] = PR[GP1:90,1] + 34.189;
   1:  PR[GP1:91,2] = PR[GP1:90,2] + -36.575;
   1:L PR[91] R[100]mm/sec CNT100;
   1:  PR[GP1:91,1] = PR[GP1:90,1] + 37.192;
   1:  PR[GP1:91,2] = PR[GP1:90,2] + -35.392;
   1:L PR[91] R[100]mm/sec CNT100;
   1:  PR[GP1:91,1] = PR[GP1:90,1] + 44.581;
   1:  PR[GP1:91,2] = PR[GP1:90,2] + -32.774;
   1:L PR[91] R[100]mm/sec CNT100;
   1:  PR[GP1:91,1] = PR[GP1:90,1] + 47.506;
   1:  PR[GP1:91,2] = PR[GP1:90,2] + -30.960;
   1:L PR[91] R[100]mm/sec CNT100;
   1:  PR[GP1:91,1] = PR[GP1:90,1] + 50.374;
   1:  PR[GP1:91,2] = PR[GP1:90,2] + -28.421;
   1:L PR[91] R[100]mm/sec CNT100;
   1:  PR[GP1:91,1] = PR[GP1:90,1] + 55.283;
   1:  PR[GP1:91,2] = PR[GP1:90,2] + -24.447;
   1:L PR[91] R[100]mm/sec CNT100;
   1:  PR[GP1:91,1] = PR[GP1:90,1] + 57.710;
   1:  PR[GP1:91,2] = PR[GP1:90,2] + -21.296;
   1:L PR[91] R[100]mm/sec CNT100;
   1:  PR[GP1:91,1] = PR[GP1:90,1] + 59.746;
   1:  PR[GP1:91,2] = PR[GP1:90,2] + -17.388;
   1:L PR[91] R[100]mm/sec CNT100;
   1:  PR[GP1:91,1] = PR[GP1:90,1] + 62.410;
   1:  PR[GP1:91,2] = PR[GP1:90,2] + -12.950;
   1:L PR[91] R[100]mm/sec CNT100;
   1:  PR[GP1:91,1] = PR[GP1:90,1] + 63.586;
   1:  PR[GP1:91,2] = PR[GP1:90,2] + -9.016;
   1:L PR[91] R[100]mm/sec CNT100;
   1:  PR[GP1:91,1] = PR[GP1:90,1] + 63.996;
   1:  PR[GP1:91,2] = PR[GP1:90,2] + -4.627;
   1:L PR[91] R[100]mm/sec CNT100;
   1:  PR[GP1:91,1] = PR[GP1:90,1] + 64.840;
   1:  PR[GP1:91,2] = PR[GP1:90,2] + -0.045;
   1:L PR[91] R[100]mm/sec CNT100;
   1:  PR[GP1:91,1] = PR[GP1:90,1] + 64.441;
   1:  PR[GP1:91,2] = PR[GP1:90,2] + 4.274;
   1:L PR[91] R[100]mm/sec CNT100;
   1:  PR[GP1:91,1] = PR[GP1:90,1] + 63.594;
   1:  PR[GP1:91,2] = PR[GP1:90,2] + 8.844;
   1:L PR[91] R[100]mm/sec CNT100;
   1:  PR[GP1:91,1] = PR[GP1:90,1] + 62.405;
   1:  PR[GP1:91,2] = PR[GP1:90,2] + 12.823;
   1:L PR[91] R[100]mm/sec CNT100;
   1:  PR[GP1:91,1] = PR[GP1:90,1] + 60.472;
   1:  PR[GP1:91,2] = PR[GP1:90,2] + 16.569;
   1:L PR[91] R[100]mm/sec CNT100;
   1:  PR[GP1:91,1] = PR[GP1:90,1] + 57.723;
   1:  PR[GP1:91,2] = PR[GP1:90,2] + 21.135;
   1:L PR[91] R[100]mm/sec CNT100;
   1:  PR[GP1:91,1] = PR[GP1:90,1] + 55.276;
   1:  PR[GP1:91,2] = PR[GP1:90,2] + 24.312;
   1:L PR[91] R[100]mm/sec CNT100;
   1:  PR[GP1:91,1] = PR[GP1:90,1] + 52.568;
   1:  PR[GP1:91,2] = PR[GP1:90,2] + 26.734;
   1:L PR[91] R[100]mm/sec CNT100;
   1:  PR[GP1:91,1] = PR[GP1:90,1] + 47.523;
   1:  PR[GP1:91,2] = PR[GP1:90,2] + 30.806;
   1:L PR[91] R[100]mm/sec CNT100;
   1:  PR[GP1:91,1] = PR[GP1:90,1] + 44.576;
   1:  PR[GP1:91,2] = PR[GP1:90,2] + 32.633;
   1:L PR[91] R[100]mm/sec CNT100;
   1:  PR[GP1:91,1] = PR[GP1:90,1] + 41.668;
   1:  PR[GP1:91,2] = PR[GP1:90,2] + 33.794;
   1:L PR[91] R[100]mm/sec CNT100;
   1:  PR[GP1:91,1] = PR[GP1:90,1] + 34.210;
   1:  PR[GP1:91,2] = PR[GP1:90,2] + 36.427;
   1:L PR[91] R[100]mm/sec CNT100;
   1:  PR[GP1:91,1] = PR[GP1:90,1] + 31.488;
   1:  PR[GP1:91,2] = PR[GP1:90,2] + 37.013;
   1:L PR[91] R[100]mm/sec CNT100;
   1:  PR[GP1:91,1] = PR[GP1:90,1] + 29.024;
   1:  PR[GP1:91,2] = PR[GP1:90,2] + 37.106;
   1:L PR[91] R[100]mm/sec CNT100;
   1:  PR[GP1:91,1] = PR[GP1:90,1] + 19.689;
   1:  PR[GP1:91,2] = PR[GP1:90,2] + 37.139;
   1:L PR[91] R[100]mm/sec CNT100;
   1:  PR[GP1:91,1] = PR[GP1:90,1] + 17.651;
   1:  PR[GP1:91,2] = PR[GP1:90,2] + 36.871;
   1:L PR[91] R[100]mm/sec CNT100;
   1:  PR[GP1:91,1] = PR[GP1:90,1] + 15.890;
   1:  PR[GP1:91,2] = PR[GP1:90,2] + 36.310;
   1:L PR[91] R[100]mm/sec CNT100;
   1:  PR[GP1:91,1] = PR[GP1:90,1] + 6.040;
   1:  PR[GP1:91,2] = PR[GP1:90,2] + 32.896;
   1:L PR[91] R[100]mm/sec CNT100;
   1:  PR[GP1:91,1] = PR[GP1:90,1] + 4.809;
   1:  PR[GP1:91,2] = PR[GP1:90,2] + 32.253;
   1:L PR[91] R[100]mm/sec CNT100;
   1:  PR[GP1:91,1] = PR[GP1:90,1] + 3.274;
   1:  PR[GP1:91,2] = PR[GP1:90,2] + 31.169;
   1:L PR[91] R[100]mm/sec CNT100;
   1:  PR[GP1:91,1] = PR[GP1:90,1] + 3.279;
   1:  PR[GP1:91,2] = PR[GP1:90,2] + 31.077;
   1:L PR[91] R[100]mm/sec CNT100;
   1:  PR[GP1:91,1] = PR[GP1:90,1] + 1.790;
   1:  PR[GP1:91,2] = PR[GP1:90,2] + 30.248;
   1:L PR[91] R[100]mm/sec CNT100;
   1:  ! -- Layer/Ebene 104 -- !;
   1:  PR[91] = PR[90];
   1:  PR[GP1:91,1] = PR[GP1:90,1] + -0.904;
   1:  PR[GP1:91,2] = PR[GP1:90,2] + 30.715;
   1:  PR[GP1:91,3] = PR[GP1:90,3] + 63.745;
   1:L PR[91] R[100]mm/sec CNT100;
   1:  PR[GP1:91,1] = PR[GP1:90,1] + -2.674;
   1:  PR[GP1:91,2] = PR[GP1:90,2] + 31.126;
   1:L PR[91] R[100]mm/sec CNT100;
   1:  PR[GP1:91,1] = PR[GP1:90,1] + -4.388;
   1:  PR[GP1:91,2] = PR[GP1:90,2] + 32.337;
   1:L PR[91] R[100]mm/sec CNT100;
   1:  PR[GP1:91,1] = PR[GP1:90,1] + -5.490;
   1:  PR[GP1:91,2] = PR[GP1:90,2] + 32.914;
   1:L PR[91] R[100]mm/sec CNT100;
   1:  PR[GP1:91,1] = PR[GP1:90,1] + -6.882;
   1:  PR[GP1:91,2] = PR[GP1:90,2] + 33.361;
   1:L PR[91] R[100]mm/sec CNT100;
   1:  PR[GP1:91,1] = PR[GP1:90,1] + -17.251;
   1:  PR[GP1:91,2] = PR[GP1:90,2] + 36.946;
   1:L PR[91] R[100]mm/sec CNT100;
   1:  PR[GP1:91,1] = PR[GP1:90,1] + -19.123;
   1:  PR[GP1:91,2] = PR[GP1:90,2] + 37.190;
   1:L PR[91] R[100]mm/sec CNT100;
   1:  PR[GP1:91,1] = PR[GP1:90,1] + -21.366;
   1:  PR[GP1:91,2] = PR[GP1:90,2] + 37.113;
   1:L PR[91] R[100]mm/sec CNT100;
   1:  PR[GP1:91,1] = PR[GP1:90,1] + -31.116;
   1:  PR[GP1:91,2] = PR[GP1:90,2] + 37.064;
   1:L PR[91] R[100]mm/sec CNT100;
   1:  PR[GP1:91,1] = PR[GP1:90,1] + -33.663;
   1:  PR[GP1:91,2] = PR[GP1:90,2] + 36.515;
   1:L PR[91] R[100]mm/sec CNT100;
   1:  PR[GP1:91,1] = PR[GP1:90,1] + -36.493;
   1:  PR[GP1:91,2] = PR[GP1:90,2] + 35.395;
   1:L PR[91] R[100]mm/sec CNT100;
   1:  PR[GP1:91,1] = PR[GP1:90,1] + -44.207;
   1:  PR[GP1:91,2] = PR[GP1:90,2] + 32.655;
   1:L PR[91] R[100]mm/sec CNT100;
   1:  PR[GP1:91,1] = PR[GP1:90,1] + -47.010;
   1:  PR[GP1:91,2] = PR[GP1:90,2] + 30.910;
   1:L PR[91] R[100]mm/sec CNT100;
   1:  PR[GP1:91,1] = PR[GP1:90,1] + -49.759;
   1:  PR[GP1:91,2] = PR[GP1:90,2] + 28.469;
   1:L PR[91] R[100]mm/sec CNT100;
   1:  PR[GP1:91,1] = PR[GP1:90,1] + -54.938;
   1:  PR[GP1:91,2] = PR[GP1:90,2] + 24.277;
   1:L PR[91] R[100]mm/sec CNT100;
   1:  PR[GP1:91,1] = PR[GP1:90,1] + -57.238;
   1:  PR[GP1:91,2] = PR[GP1:90,2] + 21.283;
   1:L PR[91] R[100]mm/sec CNT100;
   1:  PR[GP1:91,1] = PR[GP1:90,1] + -59.185;
   1:  PR[GP1:91,2] = PR[GP1:90,2] + 17.505;
   1:L PR[91] R[100]mm/sec CNT100;
   1:  PR[GP1:91,1] = PR[GP1:90,1] + -62.028;
   1:  PR[GP1:91,2] = PR[GP1:90,2] + 12.756;
   1:L PR[91] R[100]mm/sec CNT100;
   1:  PR[GP1:91,1] = PR[GP1:90,1] + -63.159;
   1:  PR[GP1:91,2] = PR[GP1:90,2] + 8.919;
   1:L PR[91] R[100]mm/sec CNT100;
   1:  PR[GP1:91,1] = PR[GP1:90,1] + -63.535;
   1:  PR[GP1:91,2] = PR[GP1:90,2] + 4.811;
   1:L PR[91] R[100]mm/sec CNT100;
   1:  PR[GP1:91,1] = PR[GP1:90,1] + -64.440;
   1:  PR[GP1:91,2] = PR[GP1:90,2] + -0.100;
   1:L PR[91] R[100]mm/sec CNT100;
   1:  PR[GP1:91,1] = PR[GP1:90,1] + -64.075;
   1:  PR[GP1:91,2] = PR[GP1:90,2] + -4.144;
   1:L PR[91] R[100]mm/sec CNT100;
   1:  PR[GP1:91,1] = PR[GP1:90,1] + -63.167;
   1:  PR[GP1:91,2] = PR[GP1:90,2] + -9.038;
   1:L PR[91] R[100]mm/sec CNT100;
   1:  PR[GP1:91,1] = PR[GP1:90,1] + -62.022;
   1:  PR[GP1:91,2] = PR[GP1:90,2] + -12.922;
   1:L PR[91] R[100]mm/sec CNT100;
   1:  PR[GP1:91,1] = PR[GP1:90,1] + -60.169;
   1:  PR[GP1:91,2] = PR[GP1:90,2] + -16.554;
   1:L PR[91] R[100]mm/sec CNT100;
   1:  PR[GP1:91,1] = PR[GP1:90,1] + -57.248;
   1:  PR[GP1:91,2] = PR[GP1:90,2] + -21.414;
   1:L PR[91] R[100]mm/sec CNT100;
   1:  PR[GP1:91,1] = PR[GP1:90,1] + -54.926;
   1:  PR[GP1:91,2] = PR[GP1:90,2] + -24.436;
   1:L PR[91] R[100]mm/sec CNT100;
   1:  PR[GP1:91,1] = PR[GP1:90,1] + -52.317;
   1:  PR[GP1:91,2] = PR[GP1:90,2] + -26.777;
   1:L PR[91] R[100]mm/sec CNT100;
   1:  PR[GP1:91,1] = PR[GP1:90,1] + -47.016;
   1:  PR[GP1:91,2] = PR[GP1:90,2] + -31.049;
   1:L PR[91] R[100]mm/sec CNT100;
   1:  PR[GP1:91,1] = PR[GP1:90,1] + -44.191;
   1:  PR[GP1:91,2] = PR[GP1:90,2] + -32.809;
   1:L PR[91] R[100]mm/sec CNT100;
   1:  PR[GP1:91,1] = PR[GP1:90,1] + -41.425;
   1:  PR[GP1:91,2] = PR[GP1:90,2] + -33.920;
   1:L PR[91] R[100]mm/sec CNT100;
   1:  PR[GP1:91,1] = PR[GP1:90,1] + -33.663;
   1:  PR[GP1:91,2] = PR[GP1:90,2] + -36.658;
   1:L PR[91] R[100]mm/sec CNT100;
   1:  PR[GP1:91,1] = PR[GP1:90,1] + -31.095;
   1:  PR[GP1:91,2] = PR[GP1:90,2] + -37.213;
   1:L PR[91] R[100]mm/sec CNT100;
   1:  PR[GP1:91,1] = PR[GP1:90,1] + -28.761;
   1:  PR[GP1:91,2] = PR[GP1:90,2] + -37.302;
   1:L PR[91] R[100]mm/sec CNT100;
   1:  PR[GP1:91,1] = PR[GP1:90,1] + -19.116;
   1:  PR[GP1:91,2] = PR[GP1:90,2] + -37.333;
   1:L PR[91] R[100]mm/sec CNT100;
   1:  PR[GP1:91,1] = PR[GP1:90,1] + -17.227;
   1:  PR[GP1:91,2] = PR[GP1:90,2] + -37.086;
   1:L PR[91] R[100]mm/sec CNT100;
   1:  PR[GP1:91,1] = PR[GP1:90,1] + -15.599;
   1:  PR[GP1:91,2] = PR[GP1:90,2] + -36.568;
   1:L PR[91] R[100]mm/sec CNT100;
   1:  PR[GP1:91,1] = PR[GP1:90,1] + -5.479;
   1:  PR[GP1:91,2] = PR[GP1:90,2] + -33.051;
   1:L PR[91] R[100]mm/sec CNT100;
   1:  PR[GP1:91,1] = PR[GP1:90,1] + -4.381;
   1:  PR[GP1:91,2] = PR[GP1:90,2] + -32.477;
   1:L PR[91] R[100]mm/sec CNT100;
   1:  PR[GP1:91,1] = PR[GP1:90,1] + -2.630;
   1:  PR[GP1:91,2] = PR[GP1:90,2] + -31.205;
   1:L PR[91] R[100]mm/sec CNT100;
   1:  PR[GP1:91,1] = PR[GP1:90,1] + -0.578;
   1:  PR[GP1:91,2] = PR[GP1:90,2] + -31.123;
   1:L PR[91] R[100]mm/sec CNT100;
   1:  PR[GP1:91,1] = PR[GP1:90,1] + 1.846;
   1:  PR[GP1:91,2] = PR[GP1:90,2] + -30.606;
   1:L PR[91] R[100]mm/sec CNT100;
   1:  PR[GP1:91,1] = PR[GP1:90,1] + 2.270;
   1:  PR[GP1:91,2] = PR[GP1:90,2] + -30.947;
   1:L PR[91] R[100]mm/sec CNT100;
   1:  PR[GP1:91,1] = PR[GP1:90,1] + 2.944;
   1:  PR[GP1:91,2] = PR[GP1:90,2] + -31.283;
   1:L PR[91] R[100]mm/sec CNT100;
   1:  PR[GP1:91,1] = PR[GP1:90,1] + 4.592;
   1:  PR[GP1:91,2] = PR[GP1:90,2] + -32.480;
   1:L PR[91] R[100]mm/sec CNT100;
   1:  PR[GP1:91,1] = PR[GP1:90,1] + 5.676;
   1:  PR[GP1:91,2] = PR[GP1:90,2] + -33.045;
   1:L PR[91] R[100]mm/sec CNT100;
   1:  PR[GP1:91,1] = PR[GP1:90,1] + 7.062;
   1:  PR[GP1:91,2] = PR[GP1:90,2] + -33.491;
   1:L PR[91] R[100]mm/sec CNT100;
   1:  PR[GP1:91,1] = PR[GP1:90,1] + 17.444;
   1:  PR[GP1:91,2] = PR[GP1:90,2] + -37.085;
   1:L PR[91] R[100]mm/sec CNT100;
   1:  PR[GP1:91,1] = PR[GP1:90,1] + 19.313;
   1:  PR[GP1:91,2] = PR[GP1:90,2] + -37.331;
   1:L PR[91] R[100]mm/sec CNT100;
   1:  PR[GP1:91,1] = PR[GP1:90,1] + 21.545;
   1:  PR[GP1:91,2] = PR[GP1:90,2] + -37.256;
   1:L PR[91] R[100]mm/sec CNT100;
   1:  PR[GP1:91,1] = PR[GP1:90,1] + 31.300;
   1:  PR[GP1:91,2] = PR[GP1:90,2] + -37.213;
   1:L PR[91] R[100]mm/sec CNT100;
   1:  PR[GP1:91,1] = PR[GP1:90,1] + 33.844;
   1:  PR[GP1:91,2] = PR[GP1:90,2] + -36.666;
   1:L PR[91] R[100]mm/sec CNT100;
   1:  PR[GP1:91,1] = PR[GP1:90,1] + 36.676;
   1:  PR[GP1:91,2] = PR[GP1:90,2] + -35.550;
   1:L PR[91] R[100]mm/sec CNT100;
   1:  PR[GP1:91,1] = PR[GP1:90,1] + 44.398;
   1:  PR[GP1:91,2] = PR[GP1:90,2] + -32.813;
   1:L PR[91] R[100]mm/sec CNT100;
   1:  PR[GP1:91,1] = PR[GP1:90,1] + 47.182;
   1:  PR[GP1:91,2] = PR[GP1:90,2] + -31.087;
   1:L PR[91] R[100]mm/sec CNT100;
   1:  PR[GP1:91,1] = PR[GP1:90,1] + 49.916;
   1:  PR[GP1:91,2] = PR[GP1:90,2] + -28.667;
   1:L PR[91] R[100]mm/sec CNT100;
   1:  PR[GP1:91,1] = PR[GP1:90,1] + 55.101;
   1:  PR[GP1:91,2] = PR[GP1:90,2] + -24.469;
   1:L PR[91] R[100]mm/sec CNT100;
   1:  PR[GP1:91,1] = PR[GP1:90,1] + 57.426;
   1:  PR[GP1:91,2] = PR[GP1:90,2] + -21.451;
   1:L PR[91] R[100]mm/sec CNT100;
   1:  PR[GP1:91,1] = PR[GP1:90,1] + 59.379;
   1:  PR[GP1:91,2] = PR[GP1:90,2] + -17.704;
   1:L PR[91] R[100]mm/sec CNT100;
   1:  PR[GP1:91,1] = PR[GP1:90,1] + 62.224;
   1:  PR[GP1:91,2] = PR[GP1:90,2] + -12.964;
   1:L PR[91] R[100]mm/sec CNT100;
   1:  PR[GP1:91,1] = PR[GP1:90,1] + 63.353;
   1:  PR[GP1:91,2] = PR[GP1:90,2] + -9.184;
   1:L PR[91] R[100]mm/sec CNT100;
   1:  PR[GP1:91,1] = PR[GP1:90,1] + 63.748;
   1:  PR[GP1:91,2] = PR[GP1:90,2] + -4.962;
   1:L PR[91] R[100]mm/sec CNT100;
   1:  PR[GP1:91,1] = PR[GP1:90,1] + 64.653;
   1:  PR[GP1:91,2] = PR[GP1:90,2] + -0.045;
   1:L PR[91] R[100]mm/sec CNT100;
   1:  PR[GP1:91,1] = PR[GP1:90,1] + 64.270;
   1:  PR[GP1:91,2] = PR[GP1:90,2] + 4.113;
   1:L PR[91] R[100]mm/sec CNT100;
   1:  PR[GP1:91,1] = PR[GP1:90,1] + 63.362;
   1:  PR[GP1:91,2] = PR[GP1:90,2] + 9.012;
   1:L PR[91] R[100]mm/sec CNT100;
   1:  PR[GP1:91,1] = PR[GP1:90,1] + 62.219;
   1:  PR[GP1:91,2] = PR[GP1:90,2] + 12.837;
   1:L PR[91] R[100]mm/sec CNT100;
   1:  PR[GP1:91,1] = PR[GP1:90,1] + 60.360;
   1:  PR[GP1:91,2] = PR[GP1:90,2] + 16.438;
   1:L PR[91] R[100]mm/sec CNT100;
   1:  PR[GP1:91,1] = PR[GP1:90,1] + 57.440;
   1:  PR[GP1:91,2] = PR[GP1:90,2] + 21.290;
   1:L PR[91] R[100]mm/sec CNT100;
   1:  PR[GP1:91,1] = PR[GP1:90,1] + 55.095;
   1:  PR[GP1:91,2] = PR[GP1:90,2] + 24.334;
   1:L PR[91] R[100]mm/sec CNT100;
   1:  PR[GP1:91,1] = PR[GP1:90,1] + 52.499;
   1:  PR[GP1:91,2] = PR[GP1:90,2] + 26.655;
   1:L PR[91] R[100]mm/sec CNT100;
   1:  PR[GP1:91,1] = PR[GP1:90,1] + 47.200;
   1:  PR[GP1:91,2] = PR[GP1:90,2] + 30.933;
   1:L PR[91] R[100]mm/sec CNT100;
   1:  PR[GP1:91,1] = PR[GP1:90,1] + 44.394;
   1:  PR[GP1:91,2] = PR[GP1:90,2] + 32.672;
   1:L PR[91] R[100]mm/sec CNT100;
   1:  PR[GP1:91,1] = PR[GP1:90,1] + 41.624;
   1:  PR[GP1:91,2] = PR[GP1:90,2] + 33.778;
   1:L PR[91] R[100]mm/sec CNT100;
   1:  PR[GP1:91,1] = PR[GP1:90,1] + 33.865;
   1:  PR[GP1:91,2] = PR[GP1:90,2] + 36.518;
   1:L PR[91] R[100]mm/sec CNT100;
   1:  PR[GP1:91,1] = PR[GP1:90,1] + 31.301;
   1:  PR[GP1:91,2] = PR[GP1:90,2] + 37.069;
   1:L PR[91] R[100]mm/sec CNT100;
   1:  PR[GP1:91,1] = PR[GP1:90,1] + 28.979;
   1:  PR[GP1:91,2] = PR[GP1:90,2] + 37.157;
   1:L PR[91] R[100]mm/sec CNT100;
   1:  PR[GP1:91,1] = PR[GP1:90,1] + 19.338;
   1:  PR[GP1:91,2] = PR[GP1:90,2] + 37.191;
   1:L PR[91] R[100]mm/sec CNT100;
   1:  PR[GP1:91,1] = PR[GP1:90,1] + 17.452;
   1:  PR[GP1:91,2] = PR[GP1:90,2] + 36.943;
   1:L PR[91] R[100]mm/sec CNT100;
   1:  PR[GP1:91,1] = PR[GP1:90,1] + 15.822;
   1:  PR[GP1:91,2] = PR[GP1:90,2] + 36.424;
   1:L PR[91] R[100]mm/sec CNT100;
   1:  PR[GP1:91,1] = PR[GP1:90,1] + 5.699;
   1:  PR[GP1:91,2] = PR[GP1:90,2] + 32.914;
   1:L PR[91] R[100]mm/sec CNT100;
   1:  PR[GP1:91,1] = PR[GP1:90,1] + 4.598;
   1:  PR[GP1:91,2] = PR[GP1:90,2] + 32.340;
   1:L PR[91] R[100]mm/sec CNT100;
   1:  PR[GP1:91,1] = PR[GP1:90,1] + 3.246;
   1:  PR[GP1:91,2] = PR[GP1:90,2] + 31.385;
   1:L PR[91] R[100]mm/sec CNT100;
   1:  PR[GP1:91,1] = PR[GP1:90,1] + 3.251;
   1:  PR[GP1:91,2] = PR[GP1:90,2] + 31.288;
   1:L PR[91] R[100]mm/sec CNT100;
   1:  PR[GP1:91,1] = PR[GP1:90,1] + 1.820;
   1:  PR[GP1:91,2] = PR[GP1:90,2] + 30.491;
   1:L PR[91] R[100]mm/sec CNT100;
   1:  ! -- Layer/Ebene 105 -- !;
   1:  PR[91] = PR[90];
   1:  PR[GP1:91,1] = PR[GP1:90,1] + -1.055;
   1:  PR[GP1:91,2] = PR[GP1:90,2] + 30.973;
   1:  PR[GP1:91,3] = PR[GP1:90,3] + 64.355;
   1:L PR[91] R[100]mm/sec CNT100;
   1:  PR[GP1:91,1] = PR[GP1:90,1] + -2.646;
   1:  PR[GP1:91,2] = PR[GP1:90,2] + 31.343;
   1:L PR[91] R[100]mm/sec CNT100;
   1:  PR[GP1:91,1] = PR[GP1:90,1] + -4.177;
   1:  PR[GP1:91,2] = PR[GP1:90,2] + 32.425;
   1:L PR[91] R[100]mm/sec CNT100;
   1:  PR[GP1:91,1] = PR[GP1:90,1] + -5.148;
   1:  PR[GP1:91,2] = PR[GP1:90,2] + 32.932;
   1:L PR[91] R[100]mm/sec CNT100;
   1:  PR[GP1:91,1] = PR[GP1:90,1] + -6.381;
   1:  PR[GP1:91,2] = PR[GP1:90,2] + 33.329;
   1:L PR[91] R[100]mm/sec CNT100;
   1:  PR[GP1:91,1] = PR[GP1:90,1] + -17.053;
   1:  PR[GP1:91,2] = PR[GP1:90,2] + 37.018;
   1:L PR[91] R[100]mm/sec CNT100;
   1:  PR[GP1:91,1] = PR[GP1:90,1] + -18.771;
   1:  PR[GP1:91,2] = PR[GP1:90,2] + 37.243;
   1:L PR[91] R[100]mm/sec CNT100;
   1:  PR[GP1:91,1] = PR[GP1:90,1] + -20.838;
   1:  PR[GP1:91,2] = PR[GP1:90,2] + 37.172;
   1:L PR[91] R[100]mm/sec CNT100;
   1:  PR[GP1:91,1] = PR[GP1:90,1] + -30.928;
   1:  PR[GP1:91,2] = PR[GP1:90,2] + 37.121;
   1:L PR[91] R[100]mm/sec CNT100;
   1:  PR[GP1:91,1] = PR[GP1:90,1] + -33.318;
   1:  PR[GP1:91,2] = PR[GP1:90,2] + 36.606;
   1:L PR[91] R[100]mm/sec CNT100;
   1:  PR[GP1:91,1] = PR[GP1:90,1] + -35.977;
   1:  PR[GP1:91,2] = PR[GP1:90,2] + 35.553;
   1:L PR[91] R[100]mm/sec CNT100;
   1:  PR[GP1:91,1] = PR[GP1:90,1] + -44.024;
   1:  PR[GP1:91,2] = PR[GP1:90,2] + 32.695;
   1:L PR[91] R[100]mm/sec CNT100;
   1:  PR[GP1:91,1] = PR[GP1:90,1] + -46.685;
   1:  PR[GP1:91,2] = PR[GP1:90,2] + 31.038;
   1:L PR[91] R[100]mm/sec CNT100;
   1:  PR[GP1:91,1] = PR[GP1:90,1] + -49.298;
   1:  PR[GP1:91,2] = PR[GP1:90,2] + 28.717;
   1:L PR[91] R[100]mm/sec CNT100;
   1:  PR[GP1:91,1] = PR[GP1:90,1] + -54.755;
   1:  PR[GP1:91,2] = PR[GP1:90,2] + 24.301;
   1:L PR[91] R[100]mm/sec CNT100;
   1:  PR[GP1:91,1] = PR[GP1:90,1] + -56.954;
   1:  PR[GP1:91,2] = PR[GP1:90,2] + 21.439;
   1:L PR[91] R[100]mm/sec CNT100;
   1:  PR[GP1:91,1] = PR[GP1:90,1] + -58.817;
   1:  PR[GP1:91,2] = PR[GP1:90,2] + 17.823;
   1:L PR[91] R[100]mm/sec CNT100;
   1:  PR[GP1:91,1] = PR[GP1:90,1] + -61.841;
   1:  PR[GP1:91,2] = PR[GP1:90,2] + 12.772;
   1:L PR[91] R[100]mm/sec CNT100;
   1:  PR[GP1:91,1] = PR[GP1:90,1] + -62.926;
   1:  PR[GP1:91,2] = PR[GP1:90,2] + 9.090;
   1:L PR[91] R[100]mm/sec CNT100;
   1:  PR[GP1:91,1] = PR[GP1:90,1] + -63.287;
   1:  PR[GP1:91,2] = PR[GP1:90,2] + 5.145;
   1:L PR[91] R[100]mm/sec CNT100;
   1:  PR[GP1:91,1] = PR[GP1:90,1] + -64.254;
   1:  PR[GP1:91,2] = PR[GP1:90,2] + -0.100;
   1:L PR[91] R[100]mm/sec CNT100;
   1:  PR[GP1:91,1] = PR[GP1:90,1] + -63.903;
   1:  PR[GP1:91,2] = PR[GP1:90,2] + -3.988;
   1:L PR[91] R[100]mm/sec CNT100;
   1:  PR[GP1:91,1] = PR[GP1:90,1] + -62.933;
   1:  PR[GP1:91,2] = PR[GP1:90,2] + -9.209;
   1:L PR[91] R[100]mm/sec CNT100;
   1:  PR[GP1:91,1] = PR[GP1:90,1] + -61.835;
   1:  PR[GP1:91,2] = PR[GP1:90,2] + -12.937;
   1:L PR[91] R[100]mm/sec CNT100;
   1:  PR[GP1:91,1] = PR[GP1:90,1] + -60.056;
   1:  PR[GP1:91,2] = PR[GP1:90,2] + -16.425;
   1:L PR[91] R[100]mm/sec CNT100;
   1:  PR[GP1:91,1] = PR[GP1:90,1] + -56.963;
   1:  PR[GP1:91,2] = PR[GP1:90,2] + -21.570;
   1:L PR[91] R[100]mm/sec CNT100;
   1:  PR[GP1:91,1] = PR[GP1:90,1] + -54.743;
   1:  PR[GP1:91,2] = PR[GP1:90,2] + -24.461;
   1:L PR[91] R[100]mm/sec CNT100;
   1:  PR[GP1:91,1] = PR[GP1:90,1] + -52.246;
   1:  PR[GP1:91,2] = PR[GP1:90,2] + -26.700;
   1:L PR[91] R[100]mm/sec CNT100;
   1:  PR[GP1:91,1] = PR[GP1:90,1] + -46.690;
   1:  PR[GP1:91,2] = PR[GP1:90,2] + -31.178;
   1:L PR[91] R[100]mm/sec CNT100;
   1:  PR[GP1:91,1] = PR[GP1:90,1] + -44.007;
   1:  PR[GP1:91,2] = PR[GP1:90,2] + -32.850;
   1:L PR[91] R[100]mm/sec CNT100;
   1:  PR[GP1:91,1] = PR[GP1:90,1] + -41.379;
   1:  PR[GP1:91,2] = PR[GP1:90,2] + -33.905;
   1:L PR[91] R[100]mm/sec CNT100;
   1:  PR[GP1:91,1] = PR[GP1:90,1] + -33.317;
   1:  PR[GP1:91,2] = PR[GP1:90,2] + -36.749;
   1:L PR[91] R[100]mm/sec CNT100;
   1:  PR[GP1:91,1] = PR[GP1:90,1] + -30.906;
   1:  PR[GP1:91,2] = PR[GP1:90,2] + -37.269;
   1:L PR[91] R[100]mm/sec CNT100;
   1:  PR[GP1:91,1] = PR[GP1:90,1] + -28.715;
   1:  PR[GP1:91,2] = PR[GP1:90,2] + -37.354;
   1:L PR[91] R[100]mm/sec CNT100;
   1:  PR[GP1:91,1] = PR[GP1:90,1] + -18.764;
   1:  PR[GP1:91,2] = PR[GP1:90,2] + -37.385;
   1:L PR[91] R[100]mm/sec CNT100;
   1:  PR[GP1:91,1] = PR[GP1:90,1] + -17.028;
   1:  PR[GP1:91,2] = PR[GP1:90,2] + -37.158;
   1:L PR[91] R[100]mm/sec CNT100;
   1:  PR[GP1:91,1] = PR[GP1:90,1] + -15.531;
   1:  PR[GP1:91,2] = PR[GP1:90,2] + -36.682;
   1:L PR[91] R[100]mm/sec CNT100;
   1:  PR[GP1:91,1] = PR[GP1:90,1] + -5.137;
   1:  PR[GP1:91,2] = PR[GP1:90,2] + -33.070;
   1:L PR[91] R[100]mm/sec CNT100;
   1:  PR[GP1:91,1] = PR[GP1:90,1] + -4.170;
   1:  PR[GP1:91,2] = PR[GP1:90,2] + -32.564;
   1:L PR[91] R[100]mm/sec CNT100;
   1:  PR[GP1:91,1] = PR[GP1:90,1] + -2.603;
   1:  PR[GP1:91,2] = PR[GP1:90,2] + -31.425;
   1:L PR[91] R[100]mm/sec CNT100;
   1:  PR[GP1:91,1] = PR[GP1:90,1] + -0.412;
   1:  PR[GP1:91,2] = PR[GP1:90,2] + -31.338;
   1:L PR[91] R[100]mm/sec CNT100;
   1:  PR[GP1:91,1] = PR[GP1:90,1] + 1.876;
   1:  PR[GP1:91,2] = PR[GP1:90,2] + -30.849;
   1:L PR[91] R[100]mm/sec CNT100;
   1:  PR[GP1:91,1] = PR[GP1:90,1] + 2.319;
   1:  PR[GP1:91,2] = PR[GP1:90,2] + -31.205;
   1:L PR[91] R[100]mm/sec CNT100;
   1:  PR[GP1:91,1] = PR[GP1:90,1] + 2.916;
   1:  PR[GP1:91,2] = PR[GP1:90,2] + -31.503;
   1:L PR[91] R[100]mm/sec CNT100;
   1:  PR[GP1:91,1] = PR[GP1:90,1] + 4.380;
   1:  PR[GP1:91,2] = PR[GP1:90,2] + -32.566;
   1:L PR[91] R[100]mm/sec CNT100;
   1:  PR[GP1:91,1] = PR[GP1:90,1] + 5.333;
   1:  PR[GP1:91,2] = PR[GP1:90,2] + -33.064;
   1:L PR[91] R[100]mm/sec CNT100;
   1:  PR[GP1:91,1] = PR[GP1:90,1] + 6.560;
   1:  PR[GP1:91,2] = PR[GP1:90,2] + -33.458;
   1:L PR[91] R[100]mm/sec CNT100;
   1:  PR[GP1:91,1] = PR[GP1:90,1] + 17.245;
   1:  PR[GP1:91,2] = PR[GP1:90,2] + -37.158;
   1:L PR[91] R[100]mm/sec CNT100;
   1:  PR[GP1:91,1] = PR[GP1:90,1] + 18.961;
   1:  PR[GP1:91,2] = PR[GP1:90,2] + -37.383;
   1:L PR[91] R[100]mm/sec CNT100;
   1:  PR[GP1:91,1] = PR[GP1:90,1] + 21.017;
   1:  PR[GP1:91,2] = PR[GP1:90,2] + -37.314;
   1:L PR[91] R[100]mm/sec CNT100;
   1:  PR[GP1:91,1] = PR[GP1:90,1] + 31.113;
   1:  PR[GP1:91,2] = PR[GP1:90,2] + -37.270;
   1:L PR[91] R[100]mm/sec CNT100;
   1:  PR[GP1:91,1] = PR[GP1:90,1] + 33.499;
   1:  PR[GP1:91,2] = PR[GP1:90,2] + -36.756;
   1:L PR[91] R[100]mm/sec CNT100;
   1:  PR[GP1:91,1] = PR[GP1:90,1] + 36.161;
   1:  PR[GP1:91,2] = PR[GP1:90,2] + -35.707;
   1:L PR[91] R[100]mm/sec CNT100;
   1:  PR[GP1:91,1] = PR[GP1:90,1] + 44.215;
   1:  PR[GP1:91,2] = PR[GP1:90,2] + -32.853;
   1:L PR[91] R[100]mm/sec CNT100;
   1:  PR[GP1:91,1] = PR[GP1:90,1] + 46.859;
   1:  PR[GP1:91,2] = PR[GP1:90,2] + -31.214;
   1:L PR[91] R[100]mm/sec CNT100;
   1:  PR[GP1:91,1] = PR[GP1:90,1] + 49.457;
   1:  PR[GP1:91,2] = PR[GP1:90,2] + -28.913;
   1:L PR[91] R[100]mm/sec CNT100;
   1:  PR[GP1:91,1] = PR[GP1:90,1] + 54.920;
   1:  PR[GP1:91,2] = PR[GP1:90,2] + -24.491;
   1:L PR[91] R[100]mm/sec CNT100;
   1:  PR[GP1:91,1] = PR[GP1:90,1] + 57.142;
   1:  PR[GP1:91,2] = PR[GP1:90,2] + -21.606;
   1:L PR[91] R[100]mm/sec CNT100;
   1:  PR[GP1:91,1] = PR[GP1:90,1] + 59.011;
   1:  PR[GP1:91,2] = PR[GP1:90,2] + -18.020;
   1:L PR[91] R[100]mm/sec CNT100;
   1:  PR[GP1:91,1] = PR[GP1:90,1] + 62.038;
   1:  PR[GP1:91,2] = PR[GP1:90,2] + -12.978;
   1:L PR[91] R[100]mm/sec CNT100;
   1:  PR[GP1:91,1] = PR[GP1:90,1] + 63.121;
   1:  PR[GP1:91,2] = PR[GP1:90,2] + -9.351;
   1:L PR[91] R[100]mm/sec CNT100;
   1:  PR[GP1:91,1] = PR[GP1:90,1] + 63.500;
   1:  PR[GP1:91,2] = PR[GP1:90,2] + -5.297;
   1:L PR[91] R[100]mm/sec CNT100;
   1:  PR[GP1:91,1] = PR[GP1:90,1] + 64.467;
   1:  PR[GP1:91,2] = PR[GP1:90,2] + -0.045;
   1:L PR[91] R[100]mm/sec CNT100;
   1:  PR[GP1:91,1] = PR[GP1:90,1] + 64.098;
   1:  PR[GP1:91,2] = PR[GP1:90,2] + 3.952;
   1:L PR[91] R[100]mm/sec CNT100;
   1:  PR[GP1:91,1] = PR[GP1:90,1] + 63.130;
   1:  PR[GP1:91,2] = PR[GP1:90,2] + 9.180;
   1:L PR[91] R[100]mm/sec CNT100;
   1:  PR[GP1:91,1] = PR[GP1:90,1] + 62.033;
   1:  PR[GP1:91,2] = PR[GP1:90,2] + 12.851;
   1:L PR[91] R[100]mm/sec CNT100;
   1:  PR[GP1:91,1] = PR[GP1:90,1] + 60.248;
   1:  PR[GP1:91,2] = PR[GP1:90,2] + 16.308;
   1:L PR[91] R[100]mm/sec CNT100;
   1:  PR[GP1:91,1] = PR[GP1:90,1] + 57.156;
   1:  PR[GP1:91,2] = PR[GP1:90,2] + 21.445;
   1:L PR[91] R[100]mm/sec CNT100;
   1:  PR[GP1:91,1] = PR[GP1:90,1] + 54.913;
   1:  PR[GP1:91,2] = PR[GP1:90,2] + 24.356;
   1:L PR[91] R[100]mm/sec CNT100;
   1:  PR[GP1:91,1] = PR[GP1:90,1] + 52.431;
   1:  PR[GP1:91,2] = PR[GP1:90,2] + 26.576;
   1:L PR[91] R[100]mm/sec CNT100;
   1:  PR[GP1:91,1] = PR[GP1:90,1] + 46.877;
   1:  PR[GP1:91,2] = PR[GP1:90,2] + 31.059;
   1:L PR[91] R[100]mm/sec CNT100;
   1:  PR[GP1:91,1] = PR[GP1:90,1] + 44.211;
   1:  PR[GP1:91,2] = PR[GP1:90,2] + 32.712;
   1:L PR[91] R[100]mm/sec CNT100;
   1:  PR[GP1:91,1] = PR[GP1:90,1] + 41.579;
   1:  PR[GP1:91,2] = PR[GP1:90,2] + 33.763;
   1:L PR[91] R[100]mm/sec CNT100;
   1:  PR[GP1:91,1] = PR[GP1:90,1] + 33.521;
   1:  PR[GP1:91,2] = PR[GP1:90,2] + 36.608;
   1:L PR[91] R[100]mm/sec CNT100;
   1:  PR[GP1:91,1] = PR[GP1:90,1] + 31.114;
   1:  PR[GP1:91,2] = PR[GP1:90,2] + 37.126;
   1:L PR[91] R[100]mm/sec CNT100;
   1:  PR[GP1:91,1] = PR[GP1:90,1] + 28.933;
   1:  PR[GP1:91,2] = PR[GP1:90,2] + 37.208;
   1:L PR[91] R[100]mm/sec CNT100;
   1:  PR[GP1:91,1] = PR[GP1:90,1] + 18.987;
   1:  PR[GP1:91,2] = PR[GP1:90,2] + 37.243;
   1:L PR[91] R[100]mm/sec CNT100;
   1:  PR[GP1:91,1] = PR[GP1:90,1] + 17.254;
   1:  PR[GP1:91,2] = PR[GP1:90,2] + 37.015;
   1:L PR[91] R[100]mm/sec CNT100;
   1:  PR[GP1:91,1] = PR[GP1:90,1] + 15.754;
   1:  PR[GP1:91,2] = PR[GP1:90,2] + 36.538;
   1:L PR[91] R[100]mm/sec CNT100;
   1:  PR[GP1:91,1] = PR[GP1:90,1] + 5.357;
   1:  PR[GP1:91,2] = PR[GP1:90,2] + 32.933;
   1:L PR[91] R[100]mm/sec CNT100;
   1:  PR[GP1:91,1] = PR[GP1:90,1] + 4.387;
   1:  PR[GP1:91,2] = PR[GP1:90,2] + 32.427;
   1:L PR[91] R[100]mm/sec CNT100;
   1:  PR[GP1:91,1] = PR[GP1:90,1] + 3.218;
   1:  PR[GP1:91,2] = PR[GP1:90,2] + 31.602;
   1:L PR[91] R[100]mm/sec CNT100;
   1:  PR[GP1:91,1] = PR[GP1:90,1] + 3.224;
   1:  PR[GP1:91,2] = PR[GP1:90,2] + 31.499;
   1:L PR[91] R[100]mm/sec CNT100;
   1:  PR[GP1:91,1] = PR[GP1:90,1] + 1.850;
   1:  PR[GP1:91,2] = PR[GP1:90,2] + 30.735;
   1:L PR[91] R[100]mm/sec CNT100;
   1:  ! -- Layer/Ebene 106 -- !;
   1:  PR[91] = PR[90];
   1:  PR[GP1:91,1] = PR[GP1:90,1] + -1.206;
   1:  PR[GP1:91,2] = PR[GP1:90,2] + 31.231;
   1:  PR[GP1:91,3] = PR[GP1:90,3] + 64.965;
   1:L PR[91] R[100]mm/sec CNT100;
   1:  PR[GP1:91,1] = PR[GP1:90,1] + -2.618;
   1:  PR[GP1:91,2] = PR[GP1:90,2] + 31.559;
   1:L PR[91] R[100]mm/sec CNT100;
   1:  PR[GP1:91,1] = PR[GP1:90,1] + -3.966;
   1:  PR[GP1:91,2] = PR[GP1:90,2] + 32.512;
   1:L PR[91] R[100]mm/sec CNT100;
   1:  PR[GP1:91,1] = PR[GP1:90,1] + -4.806;
   1:  PR[GP1:91,2] = PR[GP1:90,2] + 32.951;
   1:L PR[91] R[100]mm/sec CNT100;
   1:  PR[GP1:91,1] = PR[GP1:90,1] + -5.880;
   1:  PR[GP1:91,2] = PR[GP1:90,2] + 33.296;
   1:L PR[91] R[100]mm/sec CNT100;
   1:  PR[GP1:91,1] = PR[GP1:90,1] + -16.854;
   1:  PR[GP1:91,2] = PR[GP1:90,2] + 37.090;
   1:L PR[91] R[100]mm/sec CNT100;
   1:  PR[GP1:91,1] = PR[GP1:90,1] + -18.420;
   1:  PR[GP1:91,2] = PR[GP1:90,2] + 37.295;
   1:L PR[91] R[100]mm/sec CNT100;
   1:  PR[GP1:91,1] = PR[GP1:90,1] + -20.310;
   1:  PR[GP1:91,2] = PR[GP1:90,2] + 37.230;
   1:L PR[91] R[100]mm/sec CNT100;
   1:  PR[GP1:91,1] = PR[GP1:90,1] + -30.740;
   1:  PR[GP1:91,2] = PR[GP1:90,2] + 37.178;
   1:L PR[91] R[100]mm/sec CNT100;
   1:  PR[GP1:91,1] = PR[GP1:90,1] + -32.972;
   1:  PR[GP1:91,2] = PR[GP1:90,2] + 36.696;
   1:L PR[91] R[100]mm/sec CNT100;
   1:  PR[GP1:91,1] = PR[GP1:90,1] + -35.461;
   1:  PR[GP1:91,2] = PR[GP1:90,2] + 35.711;
   1:L PR[91] R[100]mm/sec CNT100;
   1:  PR[GP1:91,1] = PR[GP1:90,1] + -43.840;
   1:  PR[GP1:91,2] = PR[GP1:90,2] + 32.735;
   1:L PR[91] R[100]mm/sec CNT100;
   1:  PR[GP1:91,1] = PR[GP1:90,1] + -46.360;
   1:  PR[GP1:91,2] = PR[GP1:90,2] + 31.166;
   1:L PR[91] R[100]mm/sec CNT100;
   1:  PR[GP1:91,1] = PR[GP1:90,1] + -48.838;
   1:  PR[GP1:91,2] = PR[GP1:90,2] + 28.965;
   1:L PR[91] R[100]mm/sec CNT100;
   1:  PR[GP1:91,1] = PR[GP1:90,1] + -54.571;
   1:  PR[GP1:91,2] = PR[GP1:90,2] + 24.326;
   1:L PR[91] R[100]mm/sec CNT100;
   1:  PR[GP1:91,1] = PR[GP1:90,1] + -56.669;
   1:  PR[GP1:91,2] = PR[GP1:90,2] + 21.595;
   1:L PR[91] R[100]mm/sec CNT100;
   1:  PR[GP1:91,1] = PR[GP1:90,1] + -58.449;
   1:  PR[GP1:91,2] = PR[GP1:90,2] + 18.141;
   1:L PR[91] R[100]mm/sec CNT100;
   1:  PR[GP1:91,1] = PR[GP1:90,1] + -61.654;
   1:  PR[GP1:91,2] = PR[GP1:90,2] + 12.788;
   1:L PR[91] R[100]mm/sec CNT100;
   1:  PR[GP1:91,1] = PR[GP1:90,1] + -62.693;
   1:  PR[GP1:91,2] = PR[GP1:90,2] + 9.262;
   1:L PR[91] R[100]mm/sec CNT100;
   1:  PR[GP1:91,1] = PR[GP1:90,1] + -63.039;
   1:  PR[GP1:91,2] = PR[GP1:90,2] + 5.479;
   1:L PR[91] R[100]mm/sec CNT100;
   1:  PR[GP1:91,1] = PR[GP1:90,1] + -64.068;
   1:  PR[GP1:91,2] = PR[GP1:90,2] + -0.100;
   1:L PR[91] R[100]mm/sec CNT100;
   1:  PR[GP1:91,1] = PR[GP1:90,1] + -63.731;
   1:  PR[GP1:91,2] = PR[GP1:90,2] + -3.831;
   1:L PR[91] R[100]mm/sec CNT100;
   1:  PR[GP1:91,1] = PR[GP1:90,1] + -62.700;
   1:  PR[GP1:91,2] = PR[GP1:90,2] + -9.381;
   1:L PR[91] R[100]mm/sec CNT100;
   1:  PR[GP1:91,1] = PR[GP1:90,1] + -61.647;
   1:  PR[GP1:91,2] = PR[GP1:90,2] + -12.953;
   1:L PR[91] R[100]mm/sec CNT100;
   1:  PR[GP1:91,1] = PR[GP1:90,1] + -59.943;
   1:  PR[GP1:91,2] = PR[GP1:90,2] + -16.295;
   1:L PR[91] R[100]mm/sec CNT100;
   1:  PR[GP1:91,1] = PR[GP1:90,1] + -56.678;
   1:  PR[GP1:91,2] = PR[GP1:90,2] + -21.727;
   1:L PR[91] R[100]mm/sec CNT100;
   1:  PR[GP1:91,1] = PR[GP1:90,1] + -54.559;
   1:  PR[GP1:91,2] = PR[GP1:90,2] + -24.485;
   1:L PR[91] R[100]mm/sec CNT100;
   1:  PR[GP1:91,1] = PR[GP1:90,1] + -52.176;
   1:  PR[GP1:91,2] = PR[GP1:90,2] + -26.622;
